Omron CX-Programmer project 新規ﾌﾟﾛｼﾞｪｸﾄ (CX-Programmer 9.20)

# PLC 新規PLC1: CJ1G-H CPU43
I/O table (CPU CJ1G-CPU43H): rack 0 slot 0 CJ1W-EIP21

## Global symbols (name address type ; comment)
0.00 BOOL  ; ロットアップ
A202.01 BOOL  ; 通信命令実行可
A343.07 BOOL  ; CF異常
A343.08 BOOL  ; 書込み異常
A343.09 BOOL  ; 書込み不可
A343.11 BOOL  ; ファイル無し
A343.13 BOOL  ; 実行中
A343.14 BOOL  ; アクセス中
A343.15 BOOL  ; 認識完了
A351 CHANNEL  ; 分秒
A352 CHANNEL  ; 日時
A353 CHANNEL  ; 年月
A356.05 BOOL  ; 送信レディ(増設ユニット)
A356.06 BOOL  ; 受信完了(増設ユニット)
A392.04 BOOL  ; 通信異常
A392.05 BOOL  ; 送信レディ(CPUユニット)
A392.06 BOOL  ; 受信完了(CPUユニット)
A392.07 BOOL  ; 受信オーバーフロー
D0 CHANNEL  ; PC書き込み待ち列数
D1 CHANNEL  ; PC書込み可
D100 CHANNEL  ; 履歴1設定データ1
D1000 CHANNEL  ; 履歴10設定データ1
D1001 CHANNEL  ; 履歴10設定データ2
D1002 CHANNEL  ; 履歴10設定データ3
D1003 CHANNEL  ; 履歴10設定データ4
D1004 CHANNEL  ; 履歴10データ1
D1005 CHANNEL  ; 履歴10データ2
D1006 CHANNEL  ; 履歴10データ3
D1007 CHANNEL  ; 履歴10データ4
D1008 CHANNEL  ; 履歴10データ5
D1009 CHANNEL  ; 履歴10データ6
D101 CHANNEL  ; 履歴1設定データ2
D1010 CHANNEL  ; 履歴10データ7
D1011 CHANNEL  ; 履歴10データ8
D1012 CHANNEL  ; 履歴10データ9
D1013 CHANNEL  ; 履歴10データ10
D1014 CHANNEL  ; 履歴10データ11
D1015 CHANNEL  ; 履歴10データ12
D1016 CHANNEL  ; 履歴10データ13
D1017 CHANNEL  ; 履歴10データ14
D1018 CHANNEL  ; 履歴10データ15
D1019 CHANNEL  ; 履歴10データ16
D102 CHANNEL  ; 履歴1設定データ3
D1020 CHANNEL  ; 履歴10データ17
D1021 CHANNEL  ; 履歴10データ18
D1022 CHANNEL  ; 履歴10データ19
D1023 CHANNEL  ; 履歴10データ20
D1024 CHANNEL  ; 履歴10データ21
D1025 CHANNEL  ; 履歴10データ22
D1026 CHANNEL  ; 履歴10データ23
D1027 CHANNEL  ; 履歴10データ24
D1028 CHANNEL  ; 履歴10データ25
D1029 CHANNEL  ; 履歴10データ26
D103 CHANNEL  ; 履歴1設定データ4
D1030 CHANNEL  ; 履歴10データ27
D1031 CHANNEL  ; 履歴10データ28
D1032 CHANNEL  ; 履歴10データ29
D1033 CHANNEL  ; 履歴10データ30
D1034 CHANNEL  ; 履歴10データ31
D1035 CHANNEL  ; 履歴10データ32
D1036 CHANNEL  ; 履歴10データ33
D1037 CHANNEL  ; 履歴10データ34
D1038 CHANNEL  ; 履歴10データ35
D1039 CHANNEL  ; 履歴10データ36
D104 CHANNEL  ; 履歴1データ1
D1040 CHANNEL  ; 履歴10データ37
D1041 CHANNEL  ; 履歴10データ38
D1042 CHANNEL  ; 履歴10データ39
D1043 CHANNEL  ; 履歴10データ40
D1044 CHANNEL  ; 履歴10データ41
D1045 CHANNEL  ; 履歴10データ42
D1046 CHANNEL  ; 履歴10データ43
D1047 CHANNEL  ; 履歴10データ44
D1048 CHANNEL  ; 履歴10データ45
D1049 CHANNEL  ; 履歴10データ46
D105 CHANNEL  ; 履歴1データ2
D1050 CHANNEL  ; 履歴10データ47
D1051 CHANNEL  ; 履歴10データ48
D1052 CHANNEL  ; 履歴10データ49
D1053 CHANNEL  ; 履歴10データ50
D1054 CHANNEL  ; 履歴10データ51
D1055 CHANNEL  ; 履歴10データ52
D1056 CHANNEL  ; 履歴10データ53
D1057 CHANNEL  ; 履歴10データ54
D1058 CHANNEL  ; 履歴10データ55
D1059 CHANNEL  ; 履歴10データ56
D106 CHANNEL  ; 履歴1データ3
D1060 CHANNEL  ; 履歴10データ57
D1061 CHANNEL  ; 履歴10データ58
D1062 CHANNEL  ; 履歴10データ59
D1063 CHANNEL  ; 履歴10データ60
D1064 CHANNEL  ; 履歴10データ61
D1065 CHANNEL  ; 履歴10データ62
D1066 CHANNEL  ; 履歴10データ63
D1067 CHANNEL  ; 履歴10データ64
D1068 CHANNEL  ; 履歴10データ65
D1069 CHANNEL  ; 履歴10データ66
D107 CHANNEL  ; 履歴1データ4
D1070 CHANNEL  ; 履歴10データ67
D1071 CHANNEL  ; 履歴10データ68
D1072 CHANNEL  ; 履歴10データ69
D1073 CHANNEL  ; 履歴10データ70
D1074 CHANNEL  ; 履歴10データ71
D1075 CHANNEL  ; 履歴10データ72
D1076 CHANNEL  ; 履歴10データ73
D1077 CHANNEL  ; 履歴10データ74
D1078 CHANNEL  ; 履歴10データ75
D1079 CHANNEL  ; 履歴10データ76
D108 CHANNEL  ; 履歴1データ5
D1080 CHANNEL  ; 履歴10データ77
D1081 CHANNEL  ; 履歴10データ78
D1082 CHANNEL  ; 履歴10データ79
D1083 CHANNEL  ; 履歴10データ80
D1084 CHANNEL  ; 履歴10データ81
D1085 CHANNEL  ; 履歴10データ82
D1086 CHANNEL  ; 履歴10データ83
D1087 CHANNEL  ; 履歴10データ84
D1088 CHANNEL  ; 履歴10データ85
D1089 CHANNEL  ; 履歴10データ86
D109 CHANNEL  ; 履歴1データ6
D1090 CHANNEL  ; 履歴10データ87
D1091 CHANNEL  ; 履歴10データ88
D1092 CHANNEL  ; 履歴10データ89
D1093 CHANNEL  ; 履歴10データ90
D1094 CHANNEL  ; 履歴10データ91
D1095 CHANNEL  ; 履歴10データ92
D1096 CHANNEL  ; 履歴10データ93
D1097 CHANNEL  ; 履歴10データ94
D1098 CHANNEL  ; 履歴10データ95
D1099 CHANNEL  ; 履歴10データ96
D11 CHANNEL  ; 年ﾊﾞｲﾅﾘ
D110 CHANNEL  ; 履歴1データ7
D1100 CHANNEL  ; 履歴11設定データ1
D1101 CHANNEL  ; 履歴11設定データ2
D1102 CHANNEL  ; 履歴11設定データ3
D1103 CHANNEL  ; 履歴11設定データ4
D1104 CHANNEL  ; 履歴11データ1
D1105 CHANNEL  ; 履歴11データ2
D1106 CHANNEL  ; 履歴11データ3
D1107 CHANNEL  ; 履歴11データ4
D1108 CHANNEL  ; 履歴11データ5
D1109 CHANNEL  ; 履歴11データ6
D111 CHANNEL  ; 履歴1データ8
D1110 CHANNEL  ; 履歴11データ7
D1111 CHANNEL  ; 履歴11データ8
D1112 CHANNEL  ; 履歴11データ9
D1113 CHANNEL  ; 履歴11データ10
D1114 CHANNEL  ; 履歴11データ11
D1115 CHANNEL  ; 履歴11データ12
D1116 CHANNEL  ; 履歴11データ13
D1117 CHANNEL  ; 履歴11データ14
D1118 CHANNEL  ; 履歴11データ15
D1119 CHANNEL  ; 履歴11データ16
D112 CHANNEL  ; 履歴1データ9
D1120 CHANNEL  ; 履歴11データ17
D1121 CHANNEL  ; 履歴11データ18
D1122 CHANNEL  ; 履歴11データ19
D1123 CHANNEL  ; 履歴11データ20
D1124 CHANNEL  ; 履歴11データ21
D1125 CHANNEL  ; 履歴11データ22
D1126 CHANNEL  ; 履歴11データ23
D1127 CHANNEL  ; 履歴11データ24
D1128 CHANNEL  ; 履歴11データ25
D1129 CHANNEL  ; 履歴11データ26
D113 CHANNEL  ; 履歴1データ10
D1130 CHANNEL  ; 履歴11データ27
D1131 CHANNEL  ; 履歴11データ28
D1132 CHANNEL  ; 履歴11データ29
D1133 CHANNEL  ; 履歴11データ30
D1134 CHANNEL  ; 履歴11データ31
D1135 CHANNEL  ; 履歴11データ32
D1136 CHANNEL  ; 履歴11データ33
D1137 CHANNEL  ; 履歴11データ34
D1138 CHANNEL  ; 履歴11データ35
D1139 CHANNEL  ; 履歴11データ36
D114 CHANNEL  ; 履歴1データ11
D1140 CHANNEL  ; 履歴11データ37
D1141 CHANNEL  ; 履歴11データ38
D1142 CHANNEL  ; 履歴11データ39
D1143 CHANNEL  ; 履歴11データ40
D1144 CHANNEL  ; 履歴11データ41
D1145 CHANNEL  ; 履歴11データ42
D1146 CHANNEL  ; 履歴11データ43
D1147 CHANNEL  ; 履歴11データ44
D1148 CHANNEL  ; 履歴11データ45
D1149 CHANNEL  ; 履歴11データ46
D115 CHANNEL  ; 履歴1データ12
D1150 CHANNEL  ; 履歴11データ47
D1151 CHANNEL  ; 履歴11データ48
D1152 CHANNEL  ; 履歴11データ49
D1153 CHANNEL  ; 履歴11データ50
D1154 CHANNEL  ; 履歴11データ51
D1155 CHANNEL  ; 履歴11データ52
D1156 CHANNEL  ; 履歴11データ53
D1157 CHANNEL  ; 履歴11データ54
D1158 CHANNEL  ; 履歴11データ55
D1159 CHANNEL  ; 履歴11データ56
D116 CHANNEL  ; 履歴1データ13
D1160 CHANNEL  ; 履歴11データ57
D1161 CHANNEL  ; 履歴11データ58
D1162 CHANNEL  ; 履歴11データ59
D1163 CHANNEL  ; 履歴11データ60
D1164 CHANNEL  ; 履歴11データ61
D1165 CHANNEL  ; 履歴11データ62
D1166 CHANNEL  ; 履歴11データ63
D1167 CHANNEL  ; 履歴11データ64
D1168 CHANNEL  ; 履歴11データ65
D1169 CHANNEL  ; 履歴11データ66
D117 CHANNEL  ; 履歴1データ14
D1170 CHANNEL  ; 履歴11データ67
D1171 CHANNEL  ; 履歴11データ68
D1172 CHANNEL  ; 履歴11データ69
D1173 CHANNEL  ; 履歴11データ70
D1174 CHANNEL  ; 履歴11データ71
D1175 CHANNEL  ; 履歴11データ72
D1176 CHANNEL  ; 履歴11データ73
D1177 CHANNEL  ; 履歴11データ74
D1178 CHANNEL  ; 履歴11データ75
D1179 CHANNEL  ; 履歴11データ76
D118 CHANNEL  ; 履歴1データ15
D1180 CHANNEL  ; 履歴11データ77
D1181 CHANNEL  ; 履歴11データ78
D1182 CHANNEL  ; 履歴11データ79
D1183 CHANNEL  ; 履歴11データ80
D1184 CHANNEL  ; 履歴11データ81
D1185 CHANNEL  ; 履歴11データ82
D1186 CHANNEL  ; 履歴11データ83
D1187 CHANNEL  ; 履歴11データ84
D1188 CHANNEL  ; 履歴11データ85
D1189 CHANNEL  ; 履歴11データ86
D119 CHANNEL  ; 履歴1データ16
D1190 CHANNEL  ; 履歴11データ87
D1191 CHANNEL  ; 履歴11データ88
D1192 CHANNEL  ; 履歴11データ89
D1193 CHANNEL  ; 履歴11データ90
D1194 CHANNEL  ; 履歴11データ91
D1195 CHANNEL  ; 履歴11データ92
D1196 CHANNEL  ; 履歴11データ93
D1197 CHANNEL  ; 履歴11データ94
D1198 CHANNEL  ; 履歴11データ95
D1199 CHANNEL  ; 履歴11データ96
D12 CHANNEL  ; 月ﾊﾞｲﾅﾘ
D120 CHANNEL  ; 履歴1データ17
D1200 CHANNEL  ; 履歴12設定データ1
D1201 CHANNEL  ; 履歴12設定データ2
D1202 CHANNEL  ; 履歴12設定データ3
D1203 CHANNEL  ; 履歴12設定データ4
D1204 CHANNEL  ; 履歴12データ1
D1205 CHANNEL  ; 履歴12データ2
D1206 CHANNEL  ; 履歴12データ3
D1207 CHANNEL  ; 履歴12データ4
D1208 CHANNEL  ; 履歴12データ5
D1209 CHANNEL  ; 履歴12データ6
D121 CHANNEL  ; 履歴1データ18
D1210 CHANNEL  ; 履歴12データ7
D1211 CHANNEL  ; 履歴12データ8
D1212 CHANNEL  ; 履歴12データ9
D1213 CHANNEL  ; 履歴12データ10
D1214 CHANNEL  ; 履歴12データ11
D1215 CHANNEL  ; 履歴12データ12
D1216 CHANNEL  ; 履歴12データ13
D1217 CHANNEL  ; 履歴12データ14
D1218 CHANNEL  ; 履歴12データ15
D1219 CHANNEL  ; 履歴12データ16
D122 CHANNEL  ; 履歴1データ19
D1220 CHANNEL  ; 履歴12データ17
D1221 CHANNEL  ; 履歴12データ18
D1222 CHANNEL  ; 履歴12データ19
D1223 CHANNEL  ; 履歴12データ20
D1224 CHANNEL  ; 履歴12データ21
D1225 CHANNEL  ; 履歴12データ22
D1226 CHANNEL  ; 履歴12データ23
D1227 CHANNEL  ; 履歴12データ24
D1228 CHANNEL  ; 履歴12データ25
D1229 CHANNEL  ; 履歴12データ26
D123 CHANNEL  ; 履歴1データ20
D1230 CHANNEL  ; 履歴12データ27
D1231 CHANNEL  ; 履歴12データ28
D1232 CHANNEL  ; 履歴12データ29
D1233 CHANNEL  ; 履歴12データ30
D1234 CHANNEL  ; 履歴12データ31
D1235 CHANNEL  ; 履歴12データ32
D1236 CHANNEL  ; 履歴12データ33
D1237 CHANNEL  ; 履歴12データ34
D1238 CHANNEL  ; 履歴12データ35
D1239 CHANNEL  ; 履歴12データ36
D124 CHANNEL  ; 履歴1データ21
D1240 CHANNEL  ; 履歴12データ37
D1241 CHANNEL  ; 履歴12データ38
D1242 CHANNEL  ; 履歴12データ39
D1243 CHANNEL  ; 履歴12データ40
D1244 CHANNEL  ; 履歴12データ41
D1245 CHANNEL  ; 履歴12データ42
D1246 CHANNEL  ; 履歴12データ43
D1247 CHANNEL  ; 履歴12データ44
D1248 CHANNEL  ; 履歴12データ45
D1249 CHANNEL  ; 履歴12データ46
D125 CHANNEL  ; 履歴1データ22
D1250 CHANNEL  ; 履歴12データ47
D1251 CHANNEL  ; 履歴12データ48
D1252 CHANNEL  ; 履歴12データ49
D1253 CHANNEL  ; 履歴12データ50
D1254 CHANNEL  ; 履歴12データ51
D1255 CHANNEL  ; 履歴12データ52
D1256 CHANNEL  ; 履歴12データ53
D1257 CHANNEL  ; 履歴12データ54
D1258 CHANNEL  ; 履歴12データ55
D1259 CHANNEL  ; 履歴12データ56
D126 CHANNEL  ; 履歴1データ23
D1260 CHANNEL  ; 履歴12データ57
D1261 CHANNEL  ; 履歴12データ58
D1262 CHANNEL  ; 履歴12データ59
D1263 CHANNEL  ; 履歴12データ60
D1264 CHANNEL  ; 履歴12データ61
D1265 CHANNEL  ; 履歴12データ62
D1266 CHANNEL  ; 履歴12データ63
D1267 CHANNEL  ; 履歴12データ64
D1268 CHANNEL  ; 履歴12データ65
D1269 CHANNEL  ; 履歴12データ66
D127 CHANNEL  ; 履歴1データ24
D1270 CHANNEL  ; 履歴12データ67
D1271 CHANNEL  ; 履歴12データ68
D1272 CHANNEL  ; 履歴12データ69
D1273 CHANNEL  ; 履歴12データ70
D1274 CHANNEL  ; 履歴12データ71
D1275 CHANNEL  ; 履歴12データ72
D1276 CHANNEL  ; 履歴12データ73
D1277 CHANNEL  ; 履歴12データ74
D1278 CHANNEL  ; 履歴12データ75
D1279 CHANNEL  ; 履歴12データ76
D128 CHANNEL  ; 履歴1データ25
D1280 CHANNEL  ; 履歴12データ77
D1281 CHANNEL  ; 履歴12データ78
D1282 CHANNEL  ; 履歴12データ79
D1283 CHANNEL  ; 履歴12データ80
D1284 CHANNEL  ; 履歴12データ81
D1285 CHANNEL  ; 履歴12データ82
D1286 CHANNEL  ; 履歴12データ83
D1287 CHANNEL  ; 履歴12データ84
D1288 CHANNEL  ; 履歴12データ85
D1289 CHANNEL  ; 履歴12データ86
D129 CHANNEL  ; 履歴1データ26
D1290 CHANNEL  ; 履歴12データ87
D1291 CHANNEL  ; 履歴12データ88
D1292 CHANNEL  ; 履歴12データ89
D1293 CHANNEL  ; 履歴12データ90
D1294 CHANNEL  ; 履歴12データ91
D1295 CHANNEL  ; 履歴12データ92
D1296 CHANNEL  ; 履歴12データ93
D1297 CHANNEL  ; 履歴12データ94
D1298 CHANNEL  ; 履歴12データ95
D1299 CHANNEL  ; 履歴12データ96
D13 CHANNEL  ; 日ﾊﾞｲﾅﾘ
D130 CHANNEL  ; 履歴1データ27
D1300 CHANNEL  ; 履歴13設定データ1
D1301 CHANNEL  ; 履歴13設定データ2
D1302 CHANNEL  ; 履歴13設定データ3
D1303 CHANNEL  ; 履歴13設定データ4
D1304 CHANNEL  ; 履歴13データ1
D1305 CHANNEL  ; 履歴13データ2
D1306 CHANNEL  ; 履歴13データ3
D1307 CHANNEL  ; 履歴13データ4
D1308 CHANNEL  ; 履歴13データ5
D1309 CHANNEL  ; 履歴13データ6
D131 CHANNEL  ; 履歴1データ28
D1310 CHANNEL  ; 履歴13データ7
D1311 CHANNEL  ; 履歴13データ8
D1312 CHANNEL  ; 履歴13データ9
D1313 CHANNEL  ; 履歴13データ10
D1314 CHANNEL  ; 履歴13データ11
D1315 CHANNEL  ; 履歴13データ12
D1316 CHANNEL  ; 履歴13データ13
D1317 CHANNEL  ; 履歴13データ14
D1318 CHANNEL  ; 履歴13データ15
D1319 CHANNEL  ; 履歴13データ16
D132 CHANNEL  ; 履歴1データ29
D1320 CHANNEL  ; 履歴13データ17
D1321 CHANNEL  ; 履歴13データ18
D1322 CHANNEL  ; 履歴13データ19
D1323 CHANNEL  ; 履歴13データ20
D1324 CHANNEL  ; 履歴13データ21
D1325 CHANNEL  ; 履歴13データ22
D1326 CHANNEL  ; 履歴13データ23
D1327 CHANNEL  ; 履歴13データ24
D1328 CHANNEL  ; 履歴13データ25
D1329 CHANNEL  ; 履歴13データ26
D133 CHANNEL  ; 履歴1データ30
D1330 CHANNEL  ; 履歴13データ27
D1331 CHANNEL  ; 履歴13データ28
D1332 CHANNEL  ; 履歴13データ29
D1333 CHANNEL  ; 履歴13データ30
D1334 CHANNEL  ; 履歴13データ31
D1335 CHANNEL  ; 履歴13データ32
D1336 CHANNEL  ; 履歴13データ33
D1337 CHANNEL  ; 履歴13データ34
D1338 CHANNEL  ; 履歴13データ35
D1339 CHANNEL  ; 履歴13データ36
D134 CHANNEL  ; 履歴1データ31
D1340 CHANNEL  ; 履歴13データ37
D1341 CHANNEL  ; 履歴13データ38
D1342 CHANNEL  ; 履歴13データ39
D1343 CHANNEL  ; 履歴13データ40
D1344 CHANNEL  ; 履歴13データ41
D1345 CHANNEL  ; 履歴13データ42
D1346 CHANNEL  ; 履歴13データ43
D1347 CHANNEL  ; 履歴13データ44
D1348 CHANNEL  ; 履歴13データ45
D1349 CHANNEL  ; 履歴13データ46
D135 CHANNEL  ; 履歴1データ32
D1350 CHANNEL  ; 履歴13データ47
D1351 CHANNEL  ; 履歴13データ48
D1352 CHANNEL  ; 履歴13データ49
D1353 CHANNEL  ; 履歴13データ50
D1354 CHANNEL  ; 履歴13データ51
D1355 CHANNEL  ; 履歴13データ52
D1356 CHANNEL  ; 履歴13データ53
D1357 CHANNEL  ; 履歴13データ54
D1358 CHANNEL  ; 履歴13データ55
D1359 CHANNEL  ; 履歴13データ56
D136 CHANNEL  ; 履歴1データ33
D1360 CHANNEL  ; 履歴13データ57
D1361 CHANNEL  ; 履歴13データ58
D1362 CHANNEL  ; 履歴13データ59
D1363 CHANNEL  ; 履歴13データ60
D1364 CHANNEL  ; 履歴13データ61
D1365 CHANNEL  ; 履歴13データ62
D1366 CHANNEL  ; 履歴13データ63
D1367 CHANNEL  ; 履歴13データ64
D1368 CHANNEL  ; 履歴13データ65
D1369 CHANNEL  ; 履歴13データ66
D137 CHANNEL  ; 履歴1データ34
D1370 CHANNEL  ; 履歴13データ67
D1371 CHANNEL  ; 履歴13データ68
D1372 CHANNEL  ; 履歴13データ69
D1373 CHANNEL  ; 履歴13データ70
D1374 CHANNEL  ; 履歴13データ71
D1375 CHANNEL  ; 履歴13データ72
D1376 CHANNEL  ; 履歴13データ73
D1377 CHANNEL  ; 履歴13データ74
D1378 CHANNEL  ; 履歴13データ75
D1379 CHANNEL  ; 履歴13データ76
D138 CHANNEL  ; 履歴1データ35
D1380 CHANNEL  ; 履歴13データ77
D1381 CHANNEL  ; 履歴13データ78
D1382 CHANNEL  ; 履歴13データ79
D1383 CHANNEL  ; 履歴13データ80
D1384 CHANNEL  ; 履歴13データ81
D1385 CHANNEL  ; 履歴13データ82
D1386 CHANNEL  ; 履歴13データ83
D1387 CHANNEL  ; 履歴13データ84
D1388 CHANNEL  ; 履歴13データ85
D1389 CHANNEL  ; 履歴13データ86
D139 CHANNEL  ; 履歴1データ36
D1390 CHANNEL  ; 履歴13データ87
D1391 CHANNEL  ; 履歴13データ88
D1392 CHANNEL  ; 履歴13データ89
D1393 CHANNEL  ; 履歴13データ90
D1394 CHANNEL  ; 履歴13データ91
D1395 CHANNEL  ; 履歴13データ92
D1396 CHANNEL  ; 履歴13データ93
D1397 CHANNEL  ; 履歴13データ94
D1398 CHANNEL  ; 履歴13データ95
D1399 CHANNEL  ; 履歴13データ96
D14 CHANNEL  ; 時ﾊﾞｲﾅﾘ
D140 CHANNEL  ; 履歴1データ37
D1400 CHANNEL  ; 履歴14設定データ1
D1401 CHANNEL  ; 履歴14設定データ2
D1402 CHANNEL  ; 履歴14設定データ3
D1403 CHANNEL  ; 履歴14設定データ4
D1404 CHANNEL  ; 履歴14データ1
D1405 CHANNEL  ; 履歴14データ2
D1406 CHANNEL  ; 履歴14データ3
D1407 CHANNEL  ; 履歴14データ4
D1408 CHANNEL  ; 履歴14データ5
D1409 CHANNEL  ; 履歴14データ6
D141 CHANNEL  ; 履歴1データ38
D1410 CHANNEL  ; 履歴14データ7
D1411 CHANNEL  ; 履歴14データ8
D1412 CHANNEL  ; 履歴14データ9
D1413 CHANNEL  ; 履歴14データ10
D1414 CHANNEL  ; 履歴14データ11
D1415 CHANNEL  ; 履歴14データ12
D1416 CHANNEL  ; 履歴14データ13
D1417 CHANNEL  ; 履歴14データ14
D1418 CHANNEL  ; 履歴14データ15
D1419 CHANNEL  ; 履歴14データ16
D142 CHANNEL  ; 履歴1データ39
D1420 CHANNEL  ; 履歴14データ17
D1421 CHANNEL  ; 履歴14データ18
D1422 CHANNEL  ; 履歴14データ19
D1423 CHANNEL  ; 履歴14データ20
D1424 CHANNEL  ; 履歴14データ21
D1425 CHANNEL  ; 履歴14データ22
D1426 CHANNEL  ; 履歴14データ23
D1427 CHANNEL  ; 履歴14データ24
D1428 CHANNEL  ; 履歴14データ25
D1429 CHANNEL  ; 履歴14データ26
D143 CHANNEL  ; 履歴1データ40
D1430 CHANNEL  ; 履歴14データ27
D1431 CHANNEL  ; 履歴14データ28
D1432 CHANNEL  ; 履歴14データ29
D1433 CHANNEL  ; 履歴14データ30
D1434 CHANNEL  ; 履歴14データ31
D1435 CHANNEL  ; 履歴14データ32
D1436 CHANNEL  ; 履歴14データ33
D1437 CHANNEL  ; 履歴14データ34
D1438 CHANNEL  ; 履歴14データ35
D1439 CHANNEL  ; 履歴14データ36
D144 CHANNEL  ; 履歴1データ41
D1440 CHANNEL  ; 履歴14データ37
D1441 CHANNEL  ; 履歴14データ38
D1442 CHANNEL  ; 履歴14データ39
D1443 CHANNEL  ; 履歴14データ40
D1444 CHANNEL  ; 履歴14データ41
D1445 CHANNEL  ; 履歴14データ42
D1446 CHANNEL  ; 履歴14データ43
D1447 CHANNEL  ; 履歴14データ44
D1448 CHANNEL  ; 履歴14データ45
D1449 CHANNEL  ; 履歴14データ46
D145 CHANNEL  ; 履歴1データ42
D1450 CHANNEL  ; 履歴14データ47
D1451 CHANNEL  ; 履歴14データ48
D1452 CHANNEL  ; 履歴14データ49
D1453 CHANNEL  ; 履歴14データ50
D1454 CHANNEL  ; 履歴14データ51
D1455 CHANNEL  ; 履歴14データ52
D1456 CHANNEL  ; 履歴14データ53
D1457 CHANNEL  ; 履歴14データ54
D1458 CHANNEL  ; 履歴14データ55
D1459 CHANNEL  ; 履歴14データ56
D146 CHANNEL  ; 履歴1データ43
D1460 CHANNEL  ; 履歴14データ57
D1461 CHANNEL  ; 履歴14データ58
D1462 CHANNEL  ; 履歴14データ59
D1463 CHANNEL  ; 履歴14データ60
D1464 CHANNEL  ; 履歴14データ61
D1465 CHANNEL  ; 履歴14データ62
D1466 CHANNEL  ; 履歴14データ63
D1467 CHANNEL  ; 履歴14データ64
D1468 CHANNEL  ; 履歴14データ65
D1469 CHANNEL  ; 履歴14データ66
D147 CHANNEL  ; 履歴1データ44
D1470 CHANNEL  ; 履歴14データ67
D1471 CHANNEL  ; 履歴14データ68
D1472 CHANNEL  ; 履歴14データ69
D1473 CHANNEL  ; 履歴14データ70
D1474 CHANNEL  ; 履歴14データ71
D1475 CHANNEL  ; 履歴14データ72
D1476 CHANNEL  ; 履歴14データ73
D1477 CHANNEL  ; 履歴14データ74
D1478 CHANNEL  ; 履歴14データ75
D1479 CHANNEL  ; 履歴14データ76
D148 CHANNEL  ; 履歴1データ45
D1480 CHANNEL  ; 履歴14データ77
D1481 CHANNEL  ; 履歴14データ78
D1482 CHANNEL  ; 履歴14データ79
D1483 CHANNEL  ; 履歴14データ80
D1484 CHANNEL  ; 履歴14データ81
D1485 CHANNEL  ; 履歴14データ82
D1486 CHANNEL  ; 履歴14データ83
D1487 CHANNEL  ; 履歴14データ84
D1488 CHANNEL  ; 履歴14データ85
D1489 CHANNEL  ; 履歴14データ86
D149 CHANNEL  ; 履歴1データ46
D1490 CHANNEL  ; 履歴14データ87
D1491 CHANNEL  ; 履歴14データ88
D1492 CHANNEL  ; 履歴14データ89
D1493 CHANNEL  ; 履歴14データ90
D1494 CHANNEL  ; 履歴14データ91
D1495 CHANNEL  ; 履歴14データ92
D1496 CHANNEL  ; 履歴14データ93
D1497 CHANNEL  ; 履歴14データ94
D1498 CHANNEL  ; 履歴14データ95
D1499 CHANNEL  ; 履歴14データ96
D15 CHANNEL  ; 分ﾊﾞｲﾅﾘ
D150 CHANNEL  ; 履歴1データ47
D151 CHANNEL  ; 履歴1データ48
D152 CHANNEL  ; 履歴1データ49
D153 CHANNEL  ; 履歴1データ50
D154 CHANNEL  ; 履歴1データ51
D155 CHANNEL  ; 履歴1データ52
D156 CHANNEL  ; 履歴1データ53
D157 CHANNEL  ; 履歴1データ54
D158 CHANNEL  ; 履歴1データ55
D159 CHANNEL  ; 履歴1データ56
D16 CHANNEL  ; 秒ﾊﾞｲﾅﾘ
D160 CHANNEL  ; 履歴1データ57
D161 CHANNEL  ; 履歴1データ58
D162 CHANNEL  ; 履歴1データ59
D163 CHANNEL  ; 履歴1データ60
D164 CHANNEL  ; 履歴1データ61
D165 CHANNEL  ; 履歴1データ62
D166 CHANNEL  ; 履歴1データ63
D167 CHANNEL  ; 履歴1データ64
D168 CHANNEL  ; 履歴1データ65
D169 CHANNEL  ; 履歴1データ66
D17 CHANNEL  ; オーダー(H)
D170 CHANNEL  ; 履歴1データ67
D171 CHANNEL  ; 履歴1データ68
D172 CHANNEL  ; 履歴1データ69
D173 CHANNEL  ; 履歴1データ70
D174 CHANNEL  ; 履歴1データ71
D175 CHANNEL  ; 履歴1データ72
D176 CHANNEL  ; 履歴1データ73
D177 CHANNEL  ; 履歴1データ74
D178 CHANNEL  ; 履歴1データ75
D179 CHANNEL  ; 履歴1データ76
D18 CHANNEL  ; オーダー(L)
D180 CHANNEL  ; 履歴1データ77
D181 CHANNEL  ; 履歴1データ78
D182 CHANNEL  ; 履歴1データ79
D183 CHANNEL  ; 履歴1データ80
D184 CHANNEL  ; 履歴1データ81
D185 CHANNEL  ; 履歴1データ82
D186 CHANNEL  ; 履歴1データ83
D187 CHANNEL  ; 履歴1データ84
D188 CHANNEL  ; 履歴1データ85
D189 CHANNEL  ; 履歴1データ86
D19 CHANNEL  ; ロット(H)
D190 CHANNEL  ; 履歴1データ87
D191 CHANNEL  ; 履歴1データ88
D192 CHANNEL  ; 履歴1データ89
D193 CHANNEL  ; 履歴1データ90
D194 CHANNEL  ; 履歴1データ91
D195 CHANNEL  ; 履歴1データ92
D196 CHANNEL  ; 履歴1データ93
D197 CHANNEL  ; 履歴1データ94
D198 CHANNEL  ; 履歴1データ95
D199 CHANNEL  ; 履歴1データ96
D2 CHANNEL  ; PC完了フラグ
D20 CHANNEL  ; ロット(L)
D200 CHANNEL  ; 履歴2設定データ1
D201 CHANNEL  ; 履歴2設定データ2
D202 CHANNEL  ; 履歴2設定データ3
D203 CHANNEL  ; 履歴2設定データ4
D204 CHANNEL  ; 履歴2データ1
D205 CHANNEL  ; 履歴2データ2
D206 CHANNEL  ; 履歴2データ3
D207 CHANNEL  ; 履歴2データ4
D208 CHANNEL  ; 履歴2データ5
D209 CHANNEL  ; 履歴2データ6
D21 CHANNEL  ; 生産数(H)
D210 CHANNEL  ; 履歴2データ7
D211 CHANNEL  ; 履歴2データ8
D212 CHANNEL  ; 履歴2データ9
D213 CHANNEL  ; 履歴2データ10
D214 CHANNEL  ; 履歴2データ11
D215 CHANNEL  ; 履歴2データ12
D216 CHANNEL  ; 履歴2データ13
D217 CHANNEL  ; 履歴2データ14
D218 CHANNEL  ; 履歴2データ15
D219 CHANNEL  ; 履歴2データ16
D22 CHANNEL  ; 生産数(L)
D220 CHANNEL  ; 履歴2データ17
D221 CHANNEL  ; 履歴2データ18
D222 CHANNEL  ; 履歴2データ19
D223 CHANNEL  ; 履歴2データ20
D224 CHANNEL  ; 履歴2データ21
D225 CHANNEL  ; 履歴2データ22
D226 CHANNEL  ; 履歴2データ23
D227 CHANNEL  ; 履歴2データ24
D228 CHANNEL  ; 履歴2データ25
D229 CHANNEL  ; 履歴2データ26
D23 CHANNEL  ; 不良数
D230 CHANNEL  ; 履歴2データ27
D231 CHANNEL  ; 履歴2データ28
D232 CHANNEL  ; 履歴2データ29
D233 CHANNEL  ; 履歴2データ30
D234 CHANNEL  ; 履歴2データ31
D235 CHANNEL  ; 履歴2データ32
D236 CHANNEL  ; 履歴2データ33
D237 CHANNEL  ; 履歴2データ34
D238 CHANNEL  ; 履歴2データ35
D239 CHANNEL  ; 履歴2データ36
D24 CHANNEL  ; ランスショート
D240 CHANNEL  ; 履歴2データ37
D241 CHANNEL  ; 履歴2データ38
D242 CHANNEL  ; 履歴2データ39
D243 CHANNEL  ; 履歴2データ40
D244 CHANNEL  ; 履歴2データ41
D245 CHANNEL  ; 履歴2データ42
D246 CHANNEL  ; 履歴2データ43
D247 CHANNEL  ; 履歴2データ44
D248 CHANNEL  ; 履歴2データ45
D249 CHANNEL  ; 履歴2データ46
D25 CHANNEL  ; ヒケショート
D250 CHANNEL  ; 履歴2データ47
D251 CHANNEL  ; 履歴2データ48
D252 CHANNEL  ; 履歴2データ49
D253 CHANNEL  ; 履歴2データ50
D254 CHANNEL  ; 履歴2データ51
D255 CHANNEL  ; 履歴2データ52
D256 CHANNEL  ; 履歴2データ53
D257 CHANNEL  ; 履歴2データ54
D258 CHANNEL  ; 履歴2データ55
D259 CHANNEL  ; 履歴2データ56
D26 CHANNEL  ; 糸引き
D260 CHANNEL  ; 履歴2データ57
D2600 CHANNEL  ; 履歴1設定データ2
D261 CHANNEL  ; 履歴2データ58
D262 CHANNEL  ; 履歴2データ59
D263 CHANNEL  ; 履歴2データ60
D264 CHANNEL  ; 履歴2データ61
D265 CHANNEL  ; 履歴2データ62
D266 CHANNEL  ; 履歴2データ63
D267 CHANNEL  ; 履歴2データ64
D268 CHANNEL  ; 履歴2データ65
D269 CHANNEL  ; 履歴2データ66
D27 CHANNEL  ; 薄壁ショート
D270 CHANNEL  ; 履歴2データ67
D2700 CHANNEL  ; 履歴2設定データ2
D271 CHANNEL  ; 履歴2データ68
D272 CHANNEL  ; 履歴2データ69
D273 CHANNEL  ; 履歴2データ70
D274 CHANNEL  ; 履歴2データ71
D275 CHANNEL  ; 履歴2データ72
D276 CHANNEL  ; 履歴2データ73
D277 CHANNEL  ; 履歴2データ74
D278 CHANNEL  ; 履歴2データ75
D279 CHANNEL  ; 履歴2データ76
D280 CHANNEL  ; 履歴2データ77
D2800 CHANNEL  ; 履歴3設定データ2
D281 CHANNEL  ; 履歴2データ78
D282 CHANNEL  ; 履歴2データ79
D283 CHANNEL  ; 履歴2データ80
D284 CHANNEL  ; 履歴2データ81
D285 CHANNEL  ; 履歴2データ82
D286 CHANNEL  ; 履歴2データ83
D287 CHANNEL  ; 履歴2データ84
D288 CHANNEL  ; 履歴2データ85
D289 CHANNEL  ; 履歴2データ86
D290 CHANNEL  ; 履歴2データ87
D2900 CHANNEL  ; 履歴4設定データ2
D291 CHANNEL  ; 履歴2データ88
D292 CHANNEL  ; 履歴2データ89
D293 CHANNEL  ; 履歴2データ90
D294 CHANNEL  ; 履歴2データ91
D295 CHANNEL  ; 履歴2データ92
D296 CHANNEL  ; 履歴2データ93
D297 CHANNEL  ; 履歴2データ94
D298 CHANNEL  ; 履歴2データ95
D299 CHANNEL  ; 履歴2データ96
D300 CHANNEL  ; 履歴3設定データ1
D3000 CHANNEL  ; 履歴5設定データ2
D301 CHANNEL  ; 履歴3設定データ2
D302 CHANNEL  ; 履歴3設定データ3
D303 CHANNEL  ; 履歴3設定データ4
D304 CHANNEL  ; 履歴3データ1
D305 CHANNEL  ; 履歴3データ2
D306 CHANNEL  ; 履歴3データ3
D307 CHANNEL  ; 履歴3データ4
D308 CHANNEL  ; 履歴3データ5
D309 CHANNEL  ; 履歴3データ6
D310 CHANNEL  ; 履歴3データ7
D3100 CHANNEL  ; 履歴6設定データ2
D311 CHANNEL  ; 履歴3データ8
D312 CHANNEL  ; 履歴3データ9
D313 CHANNEL  ; 履歴3データ10
D314 CHANNEL  ; 履歴3データ11
D315 CHANNEL  ; 履歴3データ12
D316 CHANNEL  ; 履歴3データ13
D317 CHANNEL  ; 履歴3データ14
D318 CHANNEL  ; 履歴3データ15
D319 CHANNEL  ; 履歴3データ16
D320 CHANNEL  ; 履歴3データ17
D321 CHANNEL  ; 履歴3データ18
D322 CHANNEL  ; 履歴3データ19
D323 CHANNEL  ; 履歴3データ20
D324 CHANNEL  ; 履歴3データ21
D325 CHANNEL  ; 履歴3データ22
D326 CHANNEL  ; 履歴3データ23
D327 CHANNEL  ; 履歴3データ24
D328 CHANNEL  ; 履歴3データ25
D329 CHANNEL  ; 履歴3データ26
D330 CHANNEL  ; 履歴3データ27
D331 CHANNEL  ; 履歴3データ28
D332 CHANNEL  ; 履歴3データ29
D333 CHANNEL  ; 履歴3データ30
D334 CHANNEL  ; 履歴3データ31
D335 CHANNEL  ; 履歴3データ32
D336 CHANNEL  ; 履歴3データ33
D337 CHANNEL  ; 履歴3データ34
D338 CHANNEL  ; 履歴3データ35
D339 CHANNEL  ; 履歴3データ36
D340 CHANNEL  ; 履歴3データ37
D341 CHANNEL  ; 履歴3データ38
D342 CHANNEL  ; 履歴3データ39
D343 CHANNEL  ; 履歴3データ40
D344 CHANNEL  ; 履歴3データ41
D345 CHANNEL  ; 履歴3データ42
D346 CHANNEL  ; 履歴3データ43
D347 CHANNEL  ; 履歴3データ44
D348 CHANNEL  ; 履歴3データ45
D349 CHANNEL  ; 履歴3データ46
D350 CHANNEL  ; 履歴3データ47
D351 CHANNEL  ; 履歴3データ48
D352 CHANNEL  ; 履歴3データ49
D353 CHANNEL  ; 履歴3データ50
D354 CHANNEL  ; 履歴3データ51
D355 CHANNEL  ; 履歴3データ52
D356 CHANNEL  ; 履歴3データ53
D357 CHANNEL  ; 履歴3データ54
D358 CHANNEL  ; 履歴3データ55
D359 CHANNEL  ; 履歴3データ56
D360 CHANNEL  ; 履歴3データ57
D3600 CHANNEL  ; 履歴1設定データ2
D361 CHANNEL  ; 履歴3データ58
D362 CHANNEL  ; 履歴3データ59
D363 CHANNEL  ; 履歴3データ60
D364 CHANNEL  ; 履歴3データ61
D365 CHANNEL  ; 履歴3データ62
D366 CHANNEL  ; 履歴3データ63
D367 CHANNEL  ; 履歴3データ64
D368 CHANNEL  ; 履歴3データ65
D369 CHANNEL  ; 履歴3データ66
D370 CHANNEL  ; 履歴3データ67
D3700 CHANNEL  ; 履歴2設定データ2
D371 CHANNEL  ; 履歴3データ68
D372 CHANNEL  ; 履歴3データ69
D373 CHANNEL  ; 履歴3データ70
D374 CHANNEL  ; 履歴3データ71
D375 CHANNEL  ; 履歴3データ72
D376 CHANNEL  ; 履歴3データ73
D377 CHANNEL  ; 履歴3データ74
D378 CHANNEL  ; 履歴3データ75
D379 CHANNEL  ; 履歴3データ76
D380 CHANNEL  ; 履歴3データ77
D3800 CHANNEL  ; 履歴3設定データ2
D381 CHANNEL  ; 履歴3データ78
D382 CHANNEL  ; 履歴3データ79
D383 CHANNEL  ; 履歴3データ80
D384 CHANNEL  ; 履歴3データ81
D385 CHANNEL  ; 履歴3データ82
D386 CHANNEL  ; 履歴3データ83
D387 CHANNEL  ; 履歴3データ84
D388 CHANNEL  ; 履歴3データ85
D389 CHANNEL  ; 履歴3データ86
D390 CHANNEL  ; 履歴3データ87
D3900 CHANNEL  ; 履歴4設定データ2
D391 CHANNEL  ; 履歴3データ88
D392 CHANNEL  ; 履歴3データ89
D393 CHANNEL  ; 履歴3データ90
D394 CHANNEL  ; 履歴3データ91
D395 CHANNEL  ; 履歴3データ92
D396 CHANNEL  ; 履歴3データ93
D397 CHANNEL  ; 履歴3データ94
D398 CHANNEL  ; 履歴3データ95
D399 CHANNEL  ; 履歴3データ96
D400 CHANNEL  ; 履歴4設定データ1
D4000 CHANNEL  ; 履歴5設定データ2
D401 CHANNEL  ; 履歴4設定データ2
D402 CHANNEL  ; 履歴4設定データ3
D403 CHANNEL  ; 履歴4設定データ4
D404 CHANNEL  ; 履歴4データ1
D405 CHANNEL  ; 履歴4データ2
D406 CHANNEL  ; 履歴4データ3
D407 CHANNEL  ; 履歴4データ4
D408 CHANNEL  ; 履歴4データ5
D409 CHANNEL  ; 履歴4データ6
D410 CHANNEL  ; 履歴4データ7
D4100 CHANNEL  ; 履歴6設定データ2
D411 CHANNEL  ; 履歴4データ8
D412 CHANNEL  ; 履歴4データ9
D413 CHANNEL  ; 履歴4データ10
D414 CHANNEL  ; 履歴4データ11
D415 CHANNEL  ; 履歴4データ12
D416 CHANNEL  ; 履歴4データ13
D417 CHANNEL  ; 履歴4データ14
D418 CHANNEL  ; 履歴4データ15
D419 CHANNEL  ; 履歴4データ16
D420 CHANNEL  ; 履歴4データ17
D421 CHANNEL  ; 履歴4データ18
D422 CHANNEL  ; 履歴4データ19
D423 CHANNEL  ; 履歴4データ20
D424 CHANNEL  ; 履歴4データ21
D425 CHANNEL  ; 履歴4データ22
D426 CHANNEL  ; 履歴4データ23
D427 CHANNEL  ; 履歴4データ24
D428 CHANNEL  ; 履歴4データ25
D429 CHANNEL  ; 履歴4データ26
D430 CHANNEL  ; 履歴4データ27
D431 CHANNEL  ; 履歴4データ28
D432 CHANNEL  ; 履歴4データ29
D433 CHANNEL  ; 履歴4データ30
D434 CHANNEL  ; 履歴4データ31
D435 CHANNEL  ; 履歴4データ32
D436 CHANNEL  ; 履歴4データ33
D437 CHANNEL  ; 履歴4データ34
D438 CHANNEL  ; 履歴4データ35
D439 CHANNEL  ; 履歴4データ36
D440 CHANNEL  ; 履歴4データ37
D441 CHANNEL  ; 履歴4データ38
D442 CHANNEL  ; 履歴4データ39
D443 CHANNEL  ; 履歴4データ40
D444 CHANNEL  ; 履歴4データ41
D445 CHANNEL  ; 履歴4データ42
D446 CHANNEL  ; 履歴4データ43
D447 CHANNEL  ; 履歴4データ44
D448 CHANNEL  ; 履歴4データ45
D449 CHANNEL  ; 履歴4データ46
D450 CHANNEL  ; 履歴4データ47
D451 CHANNEL  ; 履歴4データ48
D452 CHANNEL  ; 履歴4データ49
D453 CHANNEL  ; 履歴4データ50
D454 CHANNEL  ; 履歴4データ51
D455 CHANNEL  ; 履歴4データ52
D456 CHANNEL  ; 履歴4データ53
D457 CHANNEL  ; 履歴4データ54
D458 CHANNEL  ; 履歴4データ55
D459 CHANNEL  ; 履歴4データ56
D460 CHANNEL  ; 履歴4データ57
D461 CHANNEL  ; 履歴4データ58
D462 CHANNEL  ; 履歴4データ59
D463 CHANNEL  ; 履歴4データ60
D464 CHANNEL  ; 履歴4データ61
D465 CHANNEL  ; 履歴4データ62
D466 CHANNEL  ; 履歴4データ63
D467 CHANNEL  ; 履歴4データ64
D468 CHANNEL  ; 履歴4データ65
D469 CHANNEL  ; 履歴4データ66
D470 CHANNEL  ; 履歴4データ67
D471 CHANNEL  ; 履歴4データ68
D472 CHANNEL  ; 履歴4データ69
D473 CHANNEL  ; 履歴4データ70
D474 CHANNEL  ; 履歴4データ71
D475 CHANNEL  ; 履歴4データ72
D476 CHANNEL  ; 履歴4データ73
D477 CHANNEL  ; 履歴4データ74
D478 CHANNEL  ; 履歴4データ75
D479 CHANNEL  ; 履歴4データ76
D480 CHANNEL  ; 履歴4データ77
D481 CHANNEL  ; 履歴4データ78
D482 CHANNEL  ; 履歴4データ79
D483 CHANNEL  ; 履歴4データ80
D484 CHANNEL  ; 履歴4データ81
D485 CHANNEL  ; 履歴4データ82
D486 CHANNEL  ; 履歴4データ83
D487 CHANNEL  ; 履歴4データ84
D488 CHANNEL  ; 履歴4データ85
D489 CHANNEL  ; 履歴4データ86
D490 CHANNEL  ; 履歴4データ87
D491 CHANNEL  ; 履歴4データ88
D492 CHANNEL  ; 履歴4データ89
D493 CHANNEL  ; 履歴4データ90
D494 CHANNEL  ; 履歴4データ91
D495 CHANNEL  ; 履歴4データ92
D496 CHANNEL  ; 履歴4データ93
D497 CHANNEL  ; 履歴4データ94
D498 CHANNEL  ; 履歴4データ95
D499 CHANNEL  ; 履歴4データ96
D500 CHANNEL  ; 履歴5設定データ1
D501 CHANNEL  ; 履歴5設定データ2
D502 CHANNEL  ; 履歴5設定データ3
D503 CHANNEL  ; 履歴5設定データ4
D504 CHANNEL  ; 履歴5データ1
D505 CHANNEL  ; 履歴5データ2
D506 CHANNEL  ; 履歴5データ3
D507 CHANNEL  ; 履歴5データ4
D508 CHANNEL  ; 履歴5データ5
D509 CHANNEL  ; 履歴5データ6
D510 CHANNEL  ; 履歴5データ7
D511 CHANNEL  ; 履歴5データ8
D512 CHANNEL  ; 履歴5データ9
D513 CHANNEL  ; 履歴5データ10
D514 CHANNEL  ; 履歴5データ11
D515 CHANNEL  ; 履歴5データ12
D516 CHANNEL  ; 履歴5データ13
D517 CHANNEL  ; 履歴5データ14
D518 CHANNEL  ; 履歴5データ15
D519 CHANNEL  ; 履歴5データ16
D520 CHANNEL  ; 履歴5データ17
D521 CHANNEL  ; 履歴5データ18
D522 CHANNEL  ; 履歴5データ19
D523 CHANNEL  ; 履歴5データ20
D524 CHANNEL  ; 履歴5データ21
D525 CHANNEL  ; 履歴5データ22
D526 CHANNEL  ; 履歴5データ23
D527 CHANNEL  ; 履歴5データ24
D528 CHANNEL  ; 履歴5データ25
D529 CHANNEL  ; 履歴5データ26
D530 CHANNEL  ; 履歴5データ27
D531 CHANNEL  ; 履歴5データ28
D532 CHANNEL  ; 履歴5データ29
D533 CHANNEL  ; 履歴5データ30
D534 CHANNEL  ; 履歴5データ31
D535 CHANNEL  ; 履歴5データ32
D536 CHANNEL  ; 履歴5データ33
D537 CHANNEL  ; 履歴5データ34
D538 CHANNEL  ; 履歴5データ35
D539 CHANNEL  ; 履歴5データ36
D540 CHANNEL  ; 履歴5データ37
D541 CHANNEL  ; 履歴5データ38
D542 CHANNEL  ; 履歴5データ39
D543 CHANNEL  ; 履歴5データ40
D544 CHANNEL  ; 履歴5データ41
D545 CHANNEL  ; 履歴5データ42
D546 CHANNEL  ; 履歴5データ43
D547 CHANNEL  ; 履歴5データ44
D548 CHANNEL  ; 履歴5データ45
D549 CHANNEL  ; 履歴5データ46
D550 CHANNEL  ; 履歴5データ47
D551 CHANNEL  ; 履歴5データ48
D552 CHANNEL  ; 履歴5データ49
D553 CHANNEL  ; 履歴5データ50
D554 CHANNEL  ; 履歴5データ51
D555 CHANNEL  ; 履歴5データ52
D556 CHANNEL  ; 履歴5データ53
D557 CHANNEL  ; 履歴5データ54
D558 CHANNEL  ; 履歴5データ55
D559 CHANNEL  ; 履歴5データ56
D560 CHANNEL  ; 履歴5データ57
D561 CHANNEL  ; 履歴5データ58
D562 CHANNEL  ; 履歴5データ59
D563 CHANNEL  ; 履歴5データ60
D564 CHANNEL  ; 履歴5データ61
D565 CHANNEL  ; 履歴5データ62
D566 CHANNEL  ; 履歴5データ63
D567 CHANNEL  ; 履歴5データ64
D568 CHANNEL  ; 履歴5データ65
D569 CHANNEL  ; 履歴5データ66
D570 CHANNEL  ; 履歴5データ67
D571 CHANNEL  ; 履歴5データ68
D572 CHANNEL  ; 履歴5データ69
D573 CHANNEL  ; 履歴5データ70
D574 CHANNEL  ; 履歴5データ71
D575 CHANNEL  ; 履歴5データ72
D576 CHANNEL  ; 履歴5データ73
D577 CHANNEL  ; 履歴5データ74
D578 CHANNEL  ; 履歴5データ75
D579 CHANNEL  ; 履歴5データ76
D580 CHANNEL  ; 履歴5データ77
D581 CHANNEL  ; 履歴5データ78
D582 CHANNEL  ; 履歴5データ79
D583 CHANNEL  ; 履歴5データ80
D584 CHANNEL  ; 履歴5データ81
D585 CHANNEL  ; 履歴5データ82
D586 CHANNEL  ; 履歴5データ83
D587 CHANNEL  ; 履歴5データ84
D588 CHANNEL  ; 履歴5データ85
D589 CHANNEL  ; 履歴5データ86
D590 CHANNEL  ; 履歴5データ87
D591 CHANNEL  ; 履歴5データ88
D592 CHANNEL  ; 履歴5データ89
D593 CHANNEL  ; 履歴5データ90
D594 CHANNEL  ; 履歴5データ91
D595 CHANNEL  ; 履歴5データ92
D596 CHANNEL  ; 履歴5データ93
D597 CHANNEL  ; 履歴5データ94
D598 CHANNEL  ; 履歴5データ95
D599 CHANNEL  ; 履歴5データ96
D6 CHANNEL  ; PC書き込み待ち列数_1
D600 CHANNEL  ; 履歴6設定データ1
D601 CHANNEL  ; 履歴6設定データ2
D602 CHANNEL  ; 履歴6設定データ3
D603 CHANNEL  ; 履歴6設定データ4
D604 CHANNEL  ; 履歴6データ1
D605 CHANNEL  ; 履歴6データ2
D606 CHANNEL  ; 履歴6データ3
D607 CHANNEL  ; 履歴6データ4
D608 CHANNEL  ; 履歴6データ5
D609 CHANNEL  ; 履歴6データ6
D610 CHANNEL  ; 履歴6データ7
D611 CHANNEL  ; 履歴6データ8
D612 CHANNEL  ; 履歴6データ9
D613 CHANNEL  ; 履歴6データ10
D614 CHANNEL  ; 履歴6データ11
D615 CHANNEL  ; 履歴6データ12
D616 CHANNEL  ; 履歴6データ13
D617 CHANNEL  ; 履歴6データ14
D618 CHANNEL  ; 履歴6データ15
D619 CHANNEL  ; 履歴6データ16
D620 CHANNEL  ; 履歴6データ17
D621 CHANNEL  ; 履歴6データ18
D622 CHANNEL  ; 履歴6データ19
D623 CHANNEL  ; 履歴6データ20
D624 CHANNEL  ; 履歴6データ21
D625 CHANNEL  ; 履歴6データ22
D626 CHANNEL  ; 履歴6データ23
D627 CHANNEL  ; 履歴6データ24
D628 CHANNEL  ; 履歴6データ25
D629 CHANNEL  ; 履歴6データ26
D630 CHANNEL  ; 履歴6データ27
D631 CHANNEL  ; 履歴6データ28
D632 CHANNEL  ; 履歴6データ29
D633 CHANNEL  ; 履歴6データ30
D634 CHANNEL  ; 履歴6データ31
D635 CHANNEL  ; 履歴6データ32
D636 CHANNEL  ; 履歴6データ33
D637 CHANNEL  ; 履歴6データ34
D638 CHANNEL  ; 履歴6データ35
D639 CHANNEL  ; 履歴6データ36
D640 CHANNEL  ; 履歴6データ37
D641 CHANNEL  ; 履歴6データ38
D642 CHANNEL  ; 履歴6データ39
D643 CHANNEL  ; 履歴6データ40
D644 CHANNEL  ; 履歴6データ41
D645 CHANNEL  ; 履歴6データ42
D646 CHANNEL  ; 履歴6データ43
D647 CHANNEL  ; 履歴6データ44
D648 CHANNEL  ; 履歴6データ45
D649 CHANNEL  ; 履歴6データ46
D650 CHANNEL  ; 履歴6データ47
D651 CHANNEL  ; 履歴6データ48
D652 CHANNEL  ; 履歴6データ49
D653 CHANNEL  ; 履歴6データ50
D654 CHANNEL  ; 履歴6データ51
D655 CHANNEL  ; 履歴6データ52
D656 CHANNEL  ; 履歴6データ53
D657 CHANNEL  ; 履歴6データ54
D658 CHANNEL  ; 履歴6データ55
D659 CHANNEL  ; 履歴6データ56
D660 CHANNEL  ; 履歴6データ57
D661 CHANNEL  ; 履歴6データ58
D662 CHANNEL  ; 履歴6データ59
D663 CHANNEL  ; 履歴6データ60
D664 CHANNEL  ; 履歴6データ61
D665 CHANNEL  ; 履歴6データ62
D666 CHANNEL  ; 履歴6データ63
D667 CHANNEL  ; 履歴6データ64
D668 CHANNEL  ; 履歴6データ65
D669 CHANNEL  ; 履歴6データ66
D670 CHANNEL  ; 履歴6データ67
D671 CHANNEL  ; 履歴6データ68
D672 CHANNEL  ; 履歴6データ69
D673 CHANNEL  ; 履歴6データ70
D674 CHANNEL  ; 履歴6データ71
D675 CHANNEL  ; 履歴6データ72
D676 CHANNEL  ; 履歴6データ73
D677 CHANNEL  ; 履歴6データ74
D678 CHANNEL  ; 履歴6データ75
D679 CHANNEL  ; 履歴6データ76
D680 CHANNEL  ; 履歴6データ77
D681 CHANNEL  ; 履歴6データ78
D682 CHANNEL  ; 履歴6データ79
D683 CHANNEL  ; 履歴6データ80
D684 CHANNEL  ; 履歴6データ81
D685 CHANNEL  ; 履歴6データ82
D686 CHANNEL  ; 履歴6データ83
D687 CHANNEL  ; 履歴6データ84
D688 CHANNEL  ; 履歴6データ85
D689 CHANNEL  ; 履歴6データ86
D690 CHANNEL  ; 履歴6データ87
D691 CHANNEL  ; 履歴6データ88
D692 CHANNEL  ; 履歴6データ89
D693 CHANNEL  ; 履歴6データ90
D694 CHANNEL  ; 履歴6データ91
D695 CHANNEL  ; 履歴6データ92
D696 CHANNEL  ; 履歴6データ93
D697 CHANNEL  ; 履歴6データ94
D698 CHANNEL  ; 履歴6データ95
D699 CHANNEL  ; 履歴6データ96
D7 CHANNEL  ; PC書き込み待ち列数_1
D700 CHANNEL  ; 履歴7設定データ1
D701 CHANNEL  ; 履歴7設定データ2
D702 CHANNEL  ; 履歴7設定データ3
D703 CHANNEL  ; 履歴7設定データ4
D704 CHANNEL  ; 履歴7データ1
D705 CHANNEL  ; 履歴7データ2
D706 CHANNEL  ; 履歴7データ3
D707 CHANNEL  ; 履歴7データ4
D708 CHANNEL  ; 履歴7データ5
D709 CHANNEL  ; 履歴7データ6
D710 CHANNEL  ; 履歴7データ7
D711 CHANNEL  ; 履歴7データ8
D712 CHANNEL  ; 履歴7データ9
D713 CHANNEL  ; 履歴7データ10
D714 CHANNEL  ; 履歴7データ11
D715 CHANNEL  ; 履歴7データ12
D716 CHANNEL  ; 履歴7データ13
D717 CHANNEL  ; 履歴7データ14
D718 CHANNEL  ; 履歴7データ15
D719 CHANNEL  ; 履歴7データ16
D720 CHANNEL  ; 履歴7データ17
D721 CHANNEL  ; 履歴7データ18
D722 CHANNEL  ; 履歴7データ19
D723 CHANNEL  ; 履歴7データ20
D724 CHANNEL  ; 履歴7データ21
D725 CHANNEL  ; 履歴7データ22
D726 CHANNEL  ; 履歴7データ23
D727 CHANNEL  ; 履歴7データ24
D728 CHANNEL  ; 履歴7データ25
D729 CHANNEL  ; 履歴7データ26
D730 CHANNEL  ; 履歴7データ27
D731 CHANNEL  ; 履歴7データ28
D732 CHANNEL  ; 履歴7データ29
D733 CHANNEL  ; 履歴7データ30
D734 CHANNEL  ; 履歴7データ31
D735 CHANNEL  ; 履歴7データ32
D736 CHANNEL  ; 履歴7データ33
D737 CHANNEL  ; 履歴7データ34
D738 CHANNEL  ; 履歴7データ35
D739 CHANNEL  ; 履歴7データ36
D740 CHANNEL  ; 履歴7データ37
D741 CHANNEL  ; 履歴7データ38
D742 CHANNEL  ; 履歴7データ39
D743 CHANNEL  ; 履歴7データ40
D744 CHANNEL  ; 履歴7データ41
D745 CHANNEL  ; 履歴7データ42
D746 CHANNEL  ; 履歴7データ43
D747 CHANNEL  ; 履歴7データ44
D748 CHANNEL  ; 履歴7データ45
D749 CHANNEL  ; 履歴7データ46
D750 CHANNEL  ; 履歴7データ47
D751 CHANNEL  ; 履歴7データ48
D752 CHANNEL  ; 履歴7データ49
D753 CHANNEL  ; 履歴7データ50
D754 CHANNEL  ; 履歴7データ51
D755 CHANNEL  ; 履歴7データ52
D756 CHANNEL  ; 履歴7データ53
D757 CHANNEL  ; 履歴7データ54
D758 CHANNEL  ; 履歴7データ55
D759 CHANNEL  ; 履歴7データ56
D760 CHANNEL  ; 履歴7データ57
D761 CHANNEL  ; 履歴7データ58
D762 CHANNEL  ; 履歴7データ59
D763 CHANNEL  ; 履歴7データ60
D764 CHANNEL  ; 履歴7データ61
D765 CHANNEL  ; 履歴7データ62
D766 CHANNEL  ; 履歴7データ63
D767 CHANNEL  ; 履歴7データ64
D768 CHANNEL  ; 履歴7データ65
D769 CHANNEL  ; 履歴7データ66
D770 CHANNEL  ; 履歴7データ67
D771 CHANNEL  ; 履歴7データ68
D772 CHANNEL  ; 履歴7データ69
D773 CHANNEL  ; 履歴7データ70
D774 CHANNEL  ; 履歴7データ71
D775 CHANNEL  ; 履歴7データ72
D776 CHANNEL  ; 履歴7データ73
D777 CHANNEL  ; 履歴7データ74
D778 CHANNEL  ; 履歴7データ75
D779 CHANNEL  ; 履歴7データ76
D780 CHANNEL  ; 履歴7データ77
D781 CHANNEL  ; 履歴7データ78
D782 CHANNEL  ; 履歴7データ79
D783 CHANNEL  ; 履歴7データ80
D784 CHANNEL  ; 履歴7データ81
D785 CHANNEL  ; 履歴7データ82
D786 CHANNEL  ; 履歴7データ83
D787 CHANNEL  ; 履歴7データ84
D788 CHANNEL  ; 履歴7データ85
D789 CHANNEL  ; 履歴7データ86
D790 CHANNEL  ; 履歴7データ87
D791 CHANNEL  ; 履歴7データ88
D792 CHANNEL  ; 履歴7データ89
D793 CHANNEL  ; 履歴7データ90
D794 CHANNEL  ; 履歴7データ91
D795 CHANNEL  ; 履歴7データ92
D796 CHANNEL  ; 履歴7データ93
D797 CHANNEL  ; 履歴7データ94
D798 CHANNEL  ; 履歴7データ95
D799 CHANNEL  ; 履歴7データ96
D800 CHANNEL  ; 履歴8設定データ1
D801 CHANNEL  ; 履歴8設定データ2
D802 CHANNEL  ; 履歴8設定データ3
D803 CHANNEL  ; 履歴8設定データ4
D804 CHANNEL  ; 履歴8データ1
D805 CHANNEL  ; 履歴8データ2
D806 CHANNEL  ; 履歴8データ3
D807 CHANNEL  ; 履歴8データ4
D808 CHANNEL  ; 履歴8データ5
D809 CHANNEL  ; 履歴8データ6
D810 CHANNEL  ; 履歴8データ7
D811 CHANNEL  ; 履歴8データ8
D812 CHANNEL  ; 履歴8データ9
D813 CHANNEL  ; 履歴8データ10
D814 CHANNEL  ; 履歴8データ11
D815 CHANNEL  ; 履歴8データ12
D816 CHANNEL  ; 履歴8データ13
D817 CHANNEL  ; 履歴8データ14
D818 CHANNEL  ; 履歴8データ15
D819 CHANNEL  ; 履歴8データ16
D820 CHANNEL  ; 履歴8データ17
D821 CHANNEL  ; 履歴8データ18
D822 CHANNEL  ; 履歴8データ19
D823 CHANNEL  ; 履歴8データ20
D824 CHANNEL  ; 履歴8データ21
D825 CHANNEL  ; 履歴8データ22
D826 CHANNEL  ; 履歴8データ23
D827 CHANNEL  ; 履歴8データ24
D828 CHANNEL  ; 履歴8データ25
D829 CHANNEL  ; 履歴8データ26
D830 CHANNEL  ; 履歴8データ27
D831 CHANNEL  ; 履歴8データ28
D832 CHANNEL  ; 履歴8データ29
D833 CHANNEL  ; 履歴8データ30
D834 CHANNEL  ; 履歴8データ31
D835 CHANNEL  ; 履歴8データ32
D836 CHANNEL  ; 履歴8データ33
D837 CHANNEL  ; 履歴8データ34
D838 CHANNEL  ; 履歴8データ35
D839 CHANNEL  ; 履歴8データ36
D840 CHANNEL  ; 履歴8データ37
D841 CHANNEL  ; 履歴8データ38
D842 CHANNEL  ; 履歴8データ39
D843 CHANNEL  ; 履歴8データ40
D844 CHANNEL  ; 履歴8データ41
D845 CHANNEL  ; 履歴8データ42
D846 CHANNEL  ; 履歴8データ43
D847 CHANNEL  ; 履歴8データ44
D848 CHANNEL  ; 履歴8データ45
D849 CHANNEL  ; 履歴8データ46
D850 CHANNEL  ; 履歴8データ47
D851 CHANNEL  ; 履歴8データ48
D852 CHANNEL  ; 履歴8データ49
D853 CHANNEL  ; 履歴8データ50
D854 CHANNEL  ; 履歴8データ51
D855 CHANNEL  ; 履歴8データ52
D856 CHANNEL  ; 履歴8データ53
D857 CHANNEL  ; 履歴8データ54
D858 CHANNEL  ; 履歴8データ55
D859 CHANNEL  ; 履歴8データ56
D860 CHANNEL  ; 履歴8データ57
D861 CHANNEL  ; 履歴8データ58
D862 CHANNEL  ; 履歴8データ59
D863 CHANNEL  ; 履歴8データ60
D864 CHANNEL  ; 履歴8データ61
D865 CHANNEL  ; 履歴8データ62
D866 CHANNEL  ; 履歴8データ63
D867 CHANNEL  ; 履歴8データ64
D868 CHANNEL  ; 履歴8データ65
D869 CHANNEL  ; 履歴8データ66
D870 CHANNEL  ; 履歴8データ67
D871 CHANNEL  ; 履歴8データ68
D872 CHANNEL  ; 履歴8データ69
D873 CHANNEL  ; 履歴8データ70
D874 CHANNEL  ; 履歴8データ71
D875 CHANNEL  ; 履歴8データ72
D876 CHANNEL  ; 履歴8データ73
D877 CHANNEL  ; 履歴8データ74
D878 CHANNEL  ; 履歴8データ75
D879 CHANNEL  ; 履歴8データ76
D880 CHANNEL  ; 履歴8データ77
D881 CHANNEL  ; 履歴8データ78
D882 CHANNEL  ; 履歴8データ79
D883 CHANNEL  ; 履歴8データ80
D884 CHANNEL  ; 履歴8データ81
D885 CHANNEL  ; 履歴8データ82
D886 CHANNEL  ; 履歴8データ83
D887 CHANNEL  ; 履歴8データ84
D888 CHANNEL  ; 履歴8データ85
D889 CHANNEL  ; 履歴8データ86
D890 CHANNEL  ; 履歴8データ87
D891 CHANNEL  ; 履歴8データ88
D892 CHANNEL  ; 履歴8データ89
D893 CHANNEL  ; 履歴8データ90
D894 CHANNEL  ; 履歴8データ91
D895 CHANNEL  ; 履歴8データ92
D896 CHANNEL  ; 履歴8データ93
D897 CHANNEL  ; 履歴8データ94
D898 CHANNEL  ; 履歴8データ95
D899 CHANNEL  ; 履歴8データ96
D900 CHANNEL  ; 履歴9設定データ1
D901 CHANNEL  ; 履歴9設定データ2
D902 CHANNEL  ; 履歴9設定データ3
D903 CHANNEL  ; 履歴9設定データ4
D904 CHANNEL  ; 履歴9データ1
D905 CHANNEL  ; 履歴9データ2
D906 CHANNEL  ; 履歴9データ3
D907 CHANNEL  ; 履歴9データ4
D908 CHANNEL  ; 履歴9データ5
D909 CHANNEL  ; 履歴9データ6
D910 CHANNEL  ; 履歴9データ7
D911 CHANNEL  ; 履歴9データ8
D912 CHANNEL  ; 履歴9データ9
D913 CHANNEL  ; 履歴9データ10
D914 CHANNEL  ; 履歴9データ11
D915 CHANNEL  ; 履歴9データ12
D916 CHANNEL  ; 履歴9データ13
D917 CHANNEL  ; 履歴9データ14
D918 CHANNEL  ; 履歴9データ15
D919 CHANNEL  ; 履歴9データ16
D920 CHANNEL  ; 履歴9データ17
D921 CHANNEL  ; 履歴9データ18
D922 CHANNEL  ; 履歴9データ19
D923 CHANNEL  ; 履歴9データ20
D924 CHANNEL  ; 履歴9データ21
D925 CHANNEL  ; 履歴9データ22
D926 CHANNEL  ; 履歴9データ23
D927 CHANNEL  ; 履歴9データ24
D928 CHANNEL  ; 履歴9データ25
D929 CHANNEL  ; 履歴9データ26
D930 CHANNEL  ; 履歴9データ27
D931 CHANNEL  ; 履歴9データ28
D932 CHANNEL  ; 履歴9データ29
D933 CHANNEL  ; 履歴9データ30
D934 CHANNEL  ; 履歴9データ31
D935 CHANNEL  ; 履歴9データ32
D936 CHANNEL  ; 履歴9データ33
D937 CHANNEL  ; 履歴9データ34
D938 CHANNEL  ; 履歴9データ35
D939 CHANNEL  ; 履歴9データ36
D940 CHANNEL  ; 履歴9データ37
D941 CHANNEL  ; 履歴9データ38
D942 CHANNEL  ; 履歴9データ39
D943 CHANNEL  ; 履歴9データ40
D944 CHANNEL  ; 履歴9データ41
D945 CHANNEL  ; 履歴9データ42
D946 CHANNEL  ; 履歴9データ43
D947 CHANNEL  ; 履歴9データ44
D948 CHANNEL  ; 履歴9データ45
D949 CHANNEL  ; 履歴9データ46
D950 CHANNEL  ; 履歴9データ47
D951 CHANNEL  ; 履歴9データ48
D952 CHANNEL  ; 履歴9データ49
D953 CHANNEL  ; 履歴9データ50
D954 CHANNEL  ; 履歴9データ51
D955 CHANNEL  ; 履歴9データ52
D956 CHANNEL  ; 履歴9データ53
D957 CHANNEL  ; 履歴9データ54
D958 CHANNEL  ; 履歴9データ55
D959 CHANNEL  ; 履歴9データ56
D960 CHANNEL  ; 履歴9データ57
D961 CHANNEL  ; 履歴9データ58
D962 CHANNEL  ; 履歴9データ59
D963 CHANNEL  ; 履歴9データ60
D964 CHANNEL  ; 履歴9データ61
D965 CHANNEL  ; 履歴9データ62
D966 CHANNEL  ; 履歴9データ63
D967 CHANNEL  ; 履歴9データ64
D968 CHANNEL  ; 履歴9データ65
D969 CHANNEL  ; 履歴9データ66
D970 CHANNEL  ; 履歴9データ67
D971 CHANNEL  ; 履歴9データ68
D972 CHANNEL  ; 履歴9データ69
D973 CHANNEL  ; 履歴9データ70
D974 CHANNEL  ; 履歴9データ71
D975 CHANNEL  ; 履歴9データ72
D976 CHANNEL  ; 履歴9データ73
D977 CHANNEL  ; 履歴9データ74
D978 CHANNEL  ; 履歴9データ75
D979 CHANNEL  ; 履歴9データ76
D980 CHANNEL  ; 履歴9データ77
D981 CHANNEL  ; 履歴9データ78
D982 CHANNEL  ; 履歴9データ79
D983 CHANNEL  ; 履歴9データ80
D984 CHANNEL  ; 履歴9データ81
D985 CHANNEL  ; 履歴9データ82
D986 CHANNEL  ; 履歴9データ83
D987 CHANNEL  ; 履歴9データ84
D988 CHANNEL  ; 履歴9データ85
D989 CHANNEL  ; 履歴9データ86
D990 CHANNEL  ; 履歴9データ87
D991 CHANNEL  ; 履歴9データ88
D992 CHANNEL  ; 履歴9データ89
D993 CHANNEL  ; 履歴9データ90
D994 CHANNEL  ; 履歴9データ91
D995 CHANNEL  ; 履歴9データ92
D996 CHANNEL  ; 履歴9データ93
D997 CHANNEL  ; 履歴9データ94
D998 CHANNEL  ; 履歴9データ95
D999 CHANNEL  ; 履歴9データ96
H0.00 BOOL  ; 履歴書込開始(PC書込禁止)
H0.01 BOOL  ; PC書込可
T0001 BOOL  ; 履歴保存処理開始
T0002 BOOL  ; PC書込み完了ディレイ
W0.00 BOOL  ; PC書き込みトリガ
W0.01 BOOL  ; 履歴保存処理開始
W0.02 BOOL  ; 前ロット履歴データ保存
W0.03 BOOL  ; 履歴保存完了
W0.04 BOOL  ; PC書出完了
W0.05 BOOL  ; 履歴PUSH完了
W0.06 BOOL  ; 書込み完了
W0.07 BOOL  ; PC読み取り完了

## Program 新規ﾌﾟﾛｸﾞﾗﾑ1 (cyclic task 0)
Local symbols
d CHANNEL

### Section 生産履歴保存_toPC

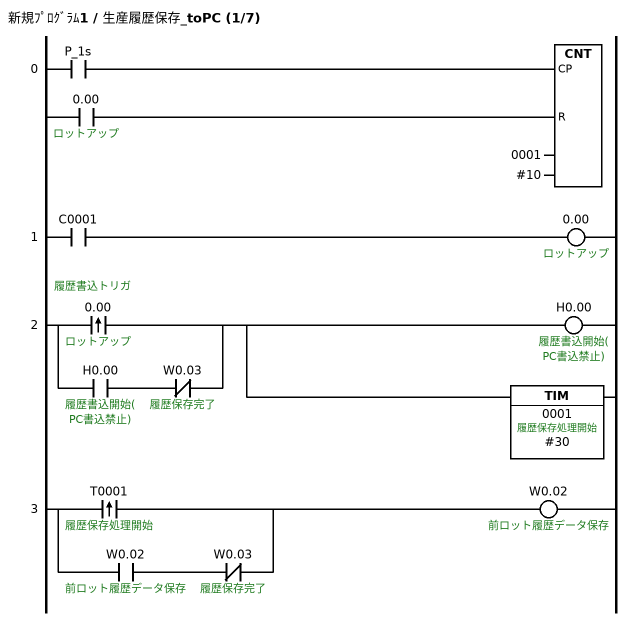
; rung 0
LD P_1s
LD 0.00  ; ロットアップ
CNT 0001 #10
; rung 1
LD C0001
OUT 0.00  ; ロットアップ
; rung 2: 履歴書込トリガ
@LD 0.00  ; ロットアップ
LD H0.00  ; 履歴書込開始(PC書込禁止)
ANDNOT W0.03  ; 履歴保存完了
ORLD
OUT H0.00  ; 履歴書込開始(PC書込禁止)
TIM 0001 #30  ; 履歴保存処理開始
; rung 3
@LD T0001  ; 履歴保存処理開始
LD W0.02  ; 前ロット履歴データ保存
ANDNOT W0.03  ; 履歴保存完了
ORLD
OUT W0.02  ; 前ロット履歴データ保存

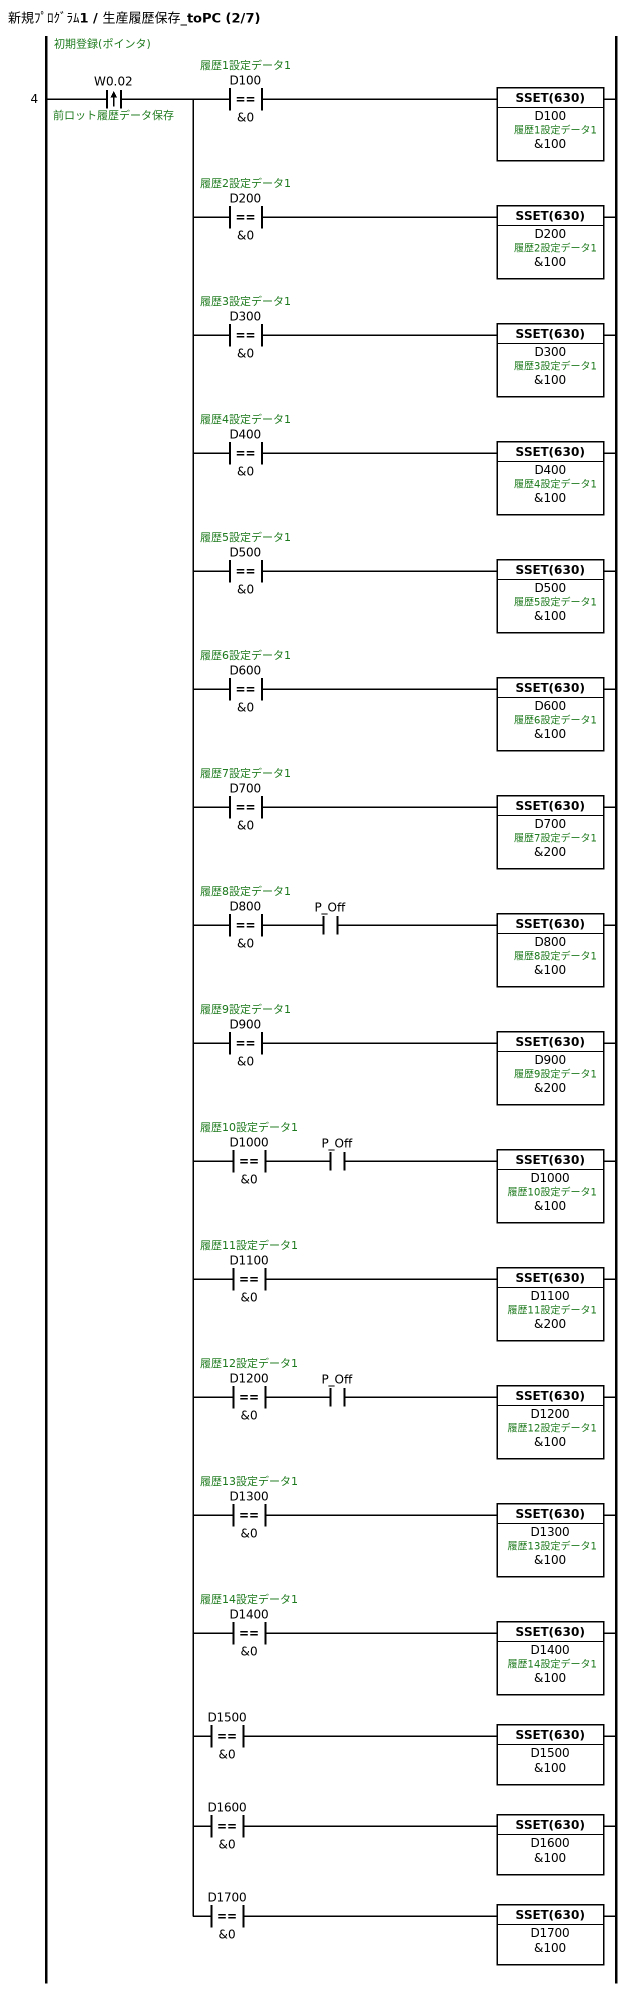
; rung 4: 初期登録(ポインタ)
@LD W0.02  ; 前ロット履歴データ保存
OUT TR0
AND=(300) D100 &0  ; 履歴1設定データ1
SSET(630) D100 &100  ; 履歴1設定データ1
LD TR0
AND=(300) D200 &0  ; 履歴2設定データ1
SSET(630) D200 &100  ; 履歴2設定データ1
LD TR0
AND=(300) D300 &0  ; 履歴3設定データ1
SSET(630) D300 &100  ; 履歴3設定データ1
LD TR0
AND=(300) D400 &0  ; 履歴4設定データ1
SSET(630) D400 &100  ; 履歴4設定データ1
LD TR0
AND=(300) D500 &0  ; 履歴5設定データ1
SSET(630) D500 &100  ; 履歴5設定データ1
LD TR0
AND=(300) D600 &0  ; 履歴6設定データ1
SSET(630) D600 &100  ; 履歴6設定データ1
LD TR0
AND=(300) D700 &0  ; 履歴7設定データ1
SSET(630) D700 &200  ; 履歴7設定データ1
LD TR0
AND=(300) D800 &0  ; 履歴8設定データ1
AND P_Off
SSET(630) D800 &100  ; 履歴8設定データ1
LD TR0
AND=(300) D900 &0  ; 履歴9設定データ1
SSET(630) D900 &200  ; 履歴9設定データ1
LD TR0
AND=(300) D1000 &0  ; 履歴10設定データ1
AND P_Off
SSET(630) D1000 &100  ; 履歴10設定データ1
LD TR0
AND=(300) D1100 &0  ; 履歴11設定データ1
SSET(630) D1100 &200  ; 履歴11設定データ1
LD TR0
AND=(300) D1200 &0  ; 履歴12設定データ1
AND P_Off
SSET(630) D1200 &100  ; 履歴12設定データ1
LD TR0
AND=(300) D1300 &0  ; 履歴13設定データ1
SSET(630) D1300 &100  ; 履歴13設定データ1
LD TR0
AND=(300) D1400 &0  ; 履歴14設定データ1
SSET(630) D1400 &100  ; 履歴14設定データ1
LD TR0
AND=(300) D1500 &0
SSET(630) D1500 &100
LD TR0
AND=(300) D1600 &0
SSET(630) D1600 &100
LD TR0
AND=(300) D1700 &0
SSET(630) D1700 &100

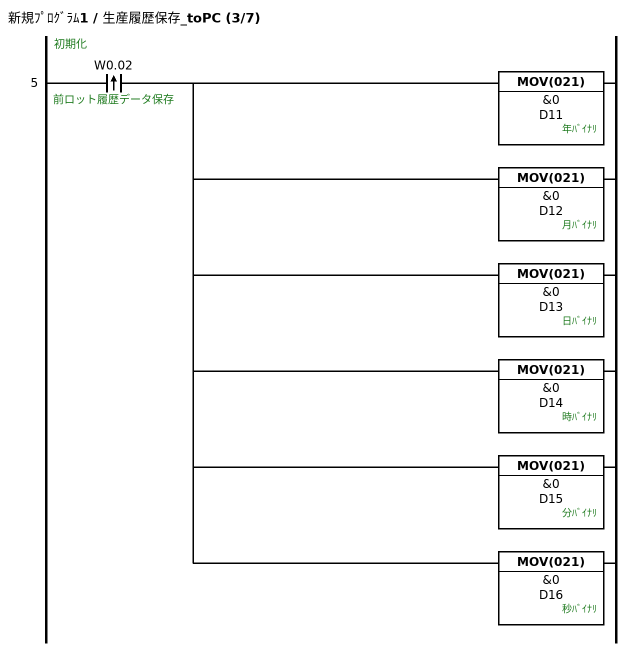
; rung 5: 初期化
@LD W0.02  ; 前ロット履歴データ保存
MOV(021) &0 D11  ; 年ﾊﾞｲﾅﾘ
MOV(021) &0 D12  ; 月ﾊﾞｲﾅﾘ
MOV(021) &0 D13  ; 日ﾊﾞｲﾅﾘ
MOV(021) &0 D14  ; 時ﾊﾞｲﾅﾘ
MOV(021) &0 D15  ; 分ﾊﾞｲﾅﾘ
MOV(021) &0 D16  ; 秒ﾊﾞｲﾅﾘ

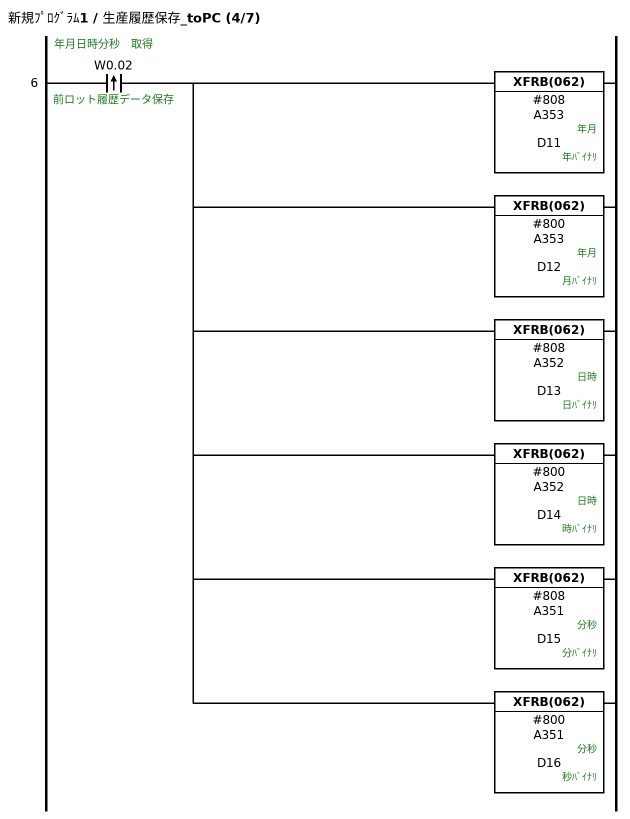
; rung 6: 年月日時分秒　取得
@LD W0.02  ; 前ロット履歴データ保存
XFRB(062) #808 A353 D11  ; 年月, 年ﾊﾞｲﾅﾘ
XFRB(062) #800 A353 D12  ; 年月, 月ﾊﾞｲﾅﾘ
XFRB(062) #808 A352 D13  ; 日時, 日ﾊﾞｲﾅﾘ
XFRB(062) #800 A352 D14  ; 日時, 時ﾊﾞｲﾅﾘ
XFRB(062) #808 A351 D15  ; 分秒, 分ﾊﾞｲﾅﾘ
XFRB(062) #800 A351 D16  ; 分秒, 秒ﾊﾞｲﾅﾘ

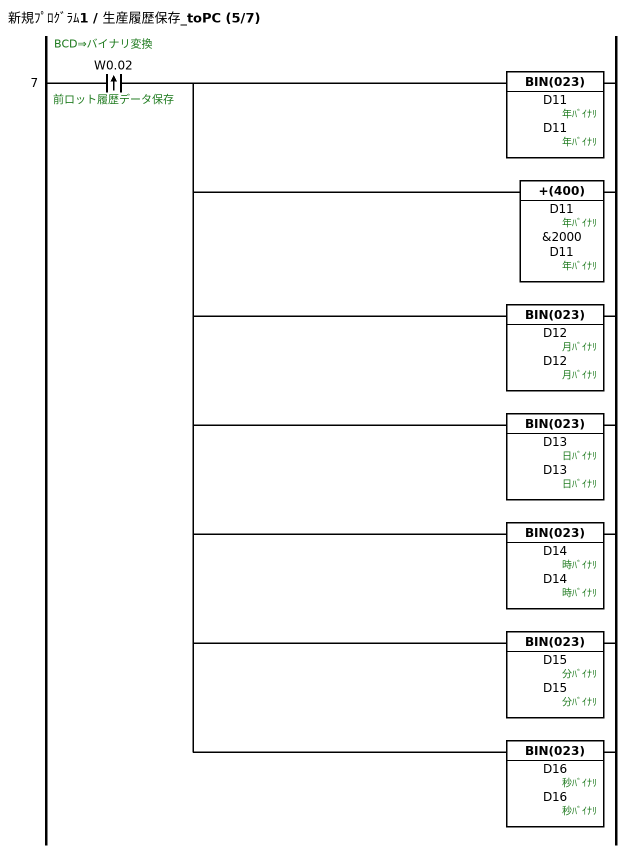
; rung 7: BCD⇒バイナリ変換
@LD W0.02  ; 前ロット履歴データ保存
BIN(023) D11 D11  ; 年ﾊﾞｲﾅﾘ
+(400) D11 &2000 D11  ; 年ﾊﾞｲﾅﾘ
BIN(023) D12 D12  ; 月ﾊﾞｲﾅﾘ
BIN(023) D13 D13  ; 日ﾊﾞｲﾅﾘ
BIN(023) D14 D14  ; 時ﾊﾞｲﾅﾘ
BIN(023) D15 D15  ; 分ﾊﾞｲﾅﾘ
BIN(023) D16 D16  ; 秒ﾊﾞｲﾅﾘ

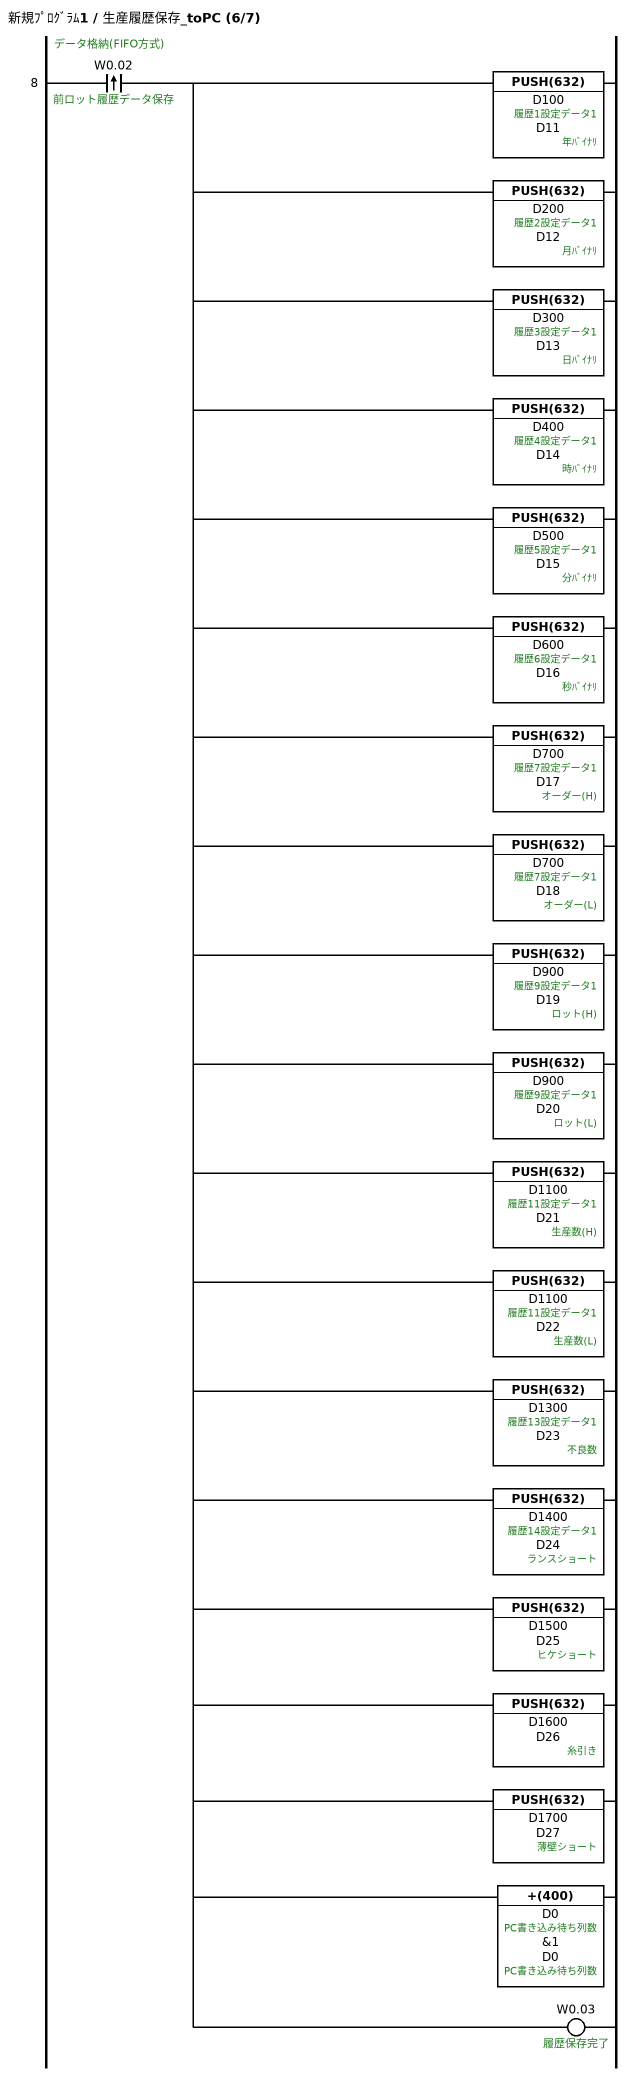
; rung 8: データ格納(FIFO方式)
@LD W0.02  ; 前ロット履歴データ保存
PUSH(632) D100 D11  ; 履歴1設定データ1, 年ﾊﾞｲﾅﾘ
PUSH(632) D200 D12  ; 履歴2設定データ1, 月ﾊﾞｲﾅﾘ
PUSH(632) D300 D13  ; 履歴3設定データ1, 日ﾊﾞｲﾅﾘ
PUSH(632) D400 D14  ; 履歴4設定データ1, 時ﾊﾞｲﾅﾘ
PUSH(632) D500 D15  ; 履歴5設定データ1, 分ﾊﾞｲﾅﾘ
PUSH(632) D600 D16  ; 履歴6設定データ1, 秒ﾊﾞｲﾅﾘ
PUSH(632) D700 D17  ; 履歴7設定データ1, オーダー(H)
PUSH(632) D700 D18  ; 履歴7設定データ1, オーダー(L)
PUSH(632) D900 D19  ; 履歴9設定データ1, ロット(H)
PUSH(632) D900 D20  ; 履歴9設定データ1, ロット(L)
PUSH(632) D1100 D21  ; 履歴11設定データ1, 生産数(H)
PUSH(632) D1100 D22  ; 履歴11設定データ1, 生産数(L)
PUSH(632) D1300 D23  ; 履歴13設定データ1, 不良数
PUSH(632) D1400 D24  ; 履歴14設定データ1, ランスショート
PUSH(632) D1500 D25  ; ヒケショート
PUSH(632) D1600 D26  ; 糸引き
PUSH(632) D1700 D27  ; 薄壁ショート
+(400) D0 &1 D0  ; PC書き込み待ち列数
OUT W0.03  ; 履歴保存完了

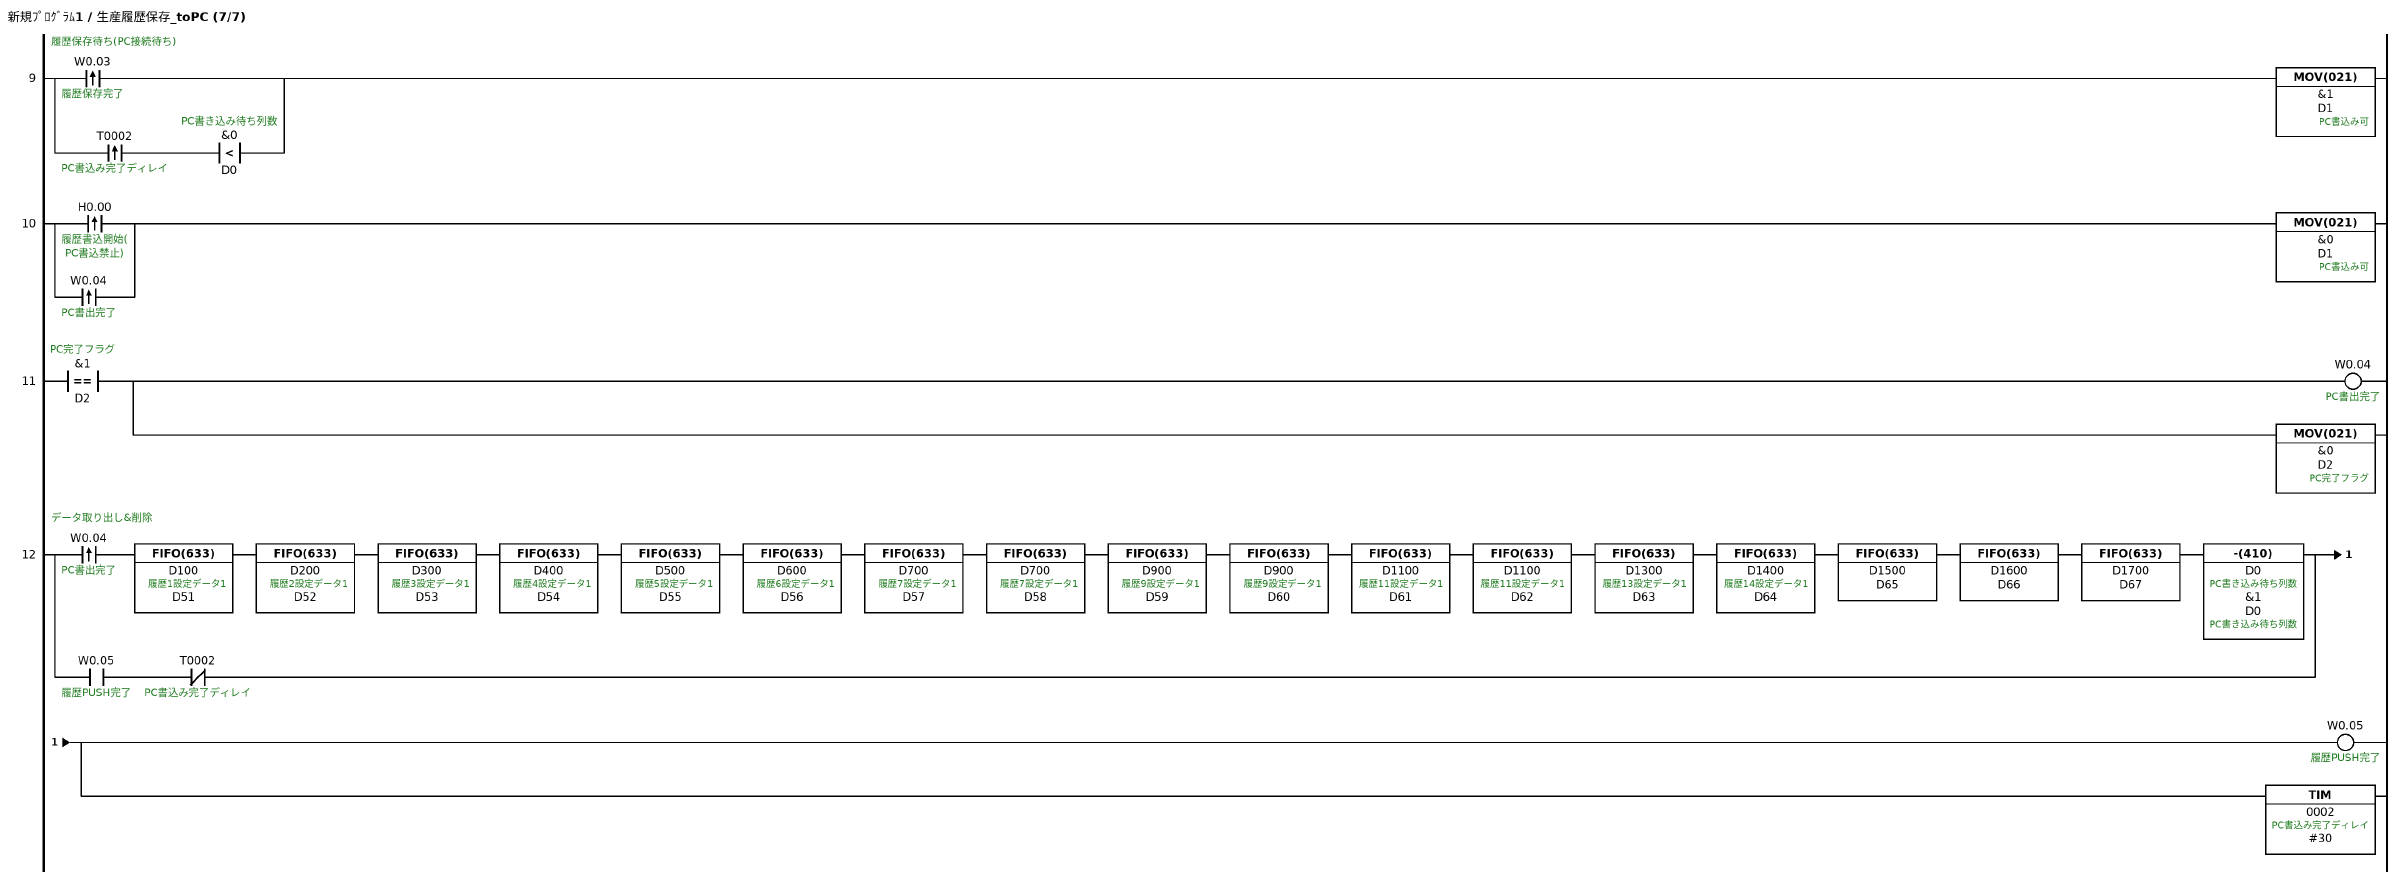
; rung 9: 履歴保存待ち(PC接続待ち)
@LD W0.03  ; 履歴保存完了
@LD T0002  ; PC書込み完了ディレイ
AND<(310) &0 D0  ; PC書き込み待ち列数
ORLD
MOV(021) &1 D1  ; PC書込み可
; rung 10
@LD H0.00  ; 履歴書込開始(PC書込禁止)
@OR W0.04  ; PC書出完了
MOV(021) &0 D1  ; PC書込み可
; rung 11
LD=(300) &1 D2  ; PC完了フラグ
OUT W0.04  ; PC書出完了
MOV(021) &0 D2  ; PC完了フラグ
; rung 12: データ取り出し&削除
@LD W0.04  ; PC書出完了
FIFO(633) D100 D51  ; 履歴1設定データ1
FIFO(633) D200 D52  ; 履歴2設定データ1
FIFO(633) D300 D53  ; 履歴3設定データ1
FIFO(633) D400 D54  ; 履歴4設定データ1
FIFO(633) D500 D55  ; 履歴5設定データ1
FIFO(633) D600 D56  ; 履歴6設定データ1
FIFO(633) D700 D57  ; 履歴7設定データ1
FIFO(633) D700 D58  ; 履歴7設定データ1
FIFO(633) D900 D59  ; 履歴9設定データ1
FIFO(633) D900 D60  ; 履歴9設定データ1
FIFO(633) D1100 D61  ; 履歴11設定データ1
FIFO(633) D1100 D62  ; 履歴11設定データ1
FIFO(633) D1300 D63  ; 履歴13設定データ1
FIFO(633) D1400 D64  ; 履歴14設定データ1
FIFO(633) D1500 D65
FIFO(633) D1600 D66
FIFO(633) D1700 D67
-(410) D0 &1 D0  ; PC書き込み待ち列数
LD W0.05  ; 履歴PUSH完了
ANDNOT T0002  ; PC書込み完了ディレイ
ORLD
OUT W0.05  ; 履歴PUSH完了
TIM 0002 #30  ; PC書込み完了ディレイ

### Section END
; rung 0
END(001)